IF state = 0 OR state = 9 THEN
	IF Busy THEN
		LastExecutionResult.Done := Done;
		LastExecutionResult.CommandAborted := CommandAborted;
		LastExecutionResult.Error := Error;
		LastExecutionResult.ErrorID := ErrorID;
	END_IF
	Busy := FALSE;
	Active := FALSE;
ELSIF F_AxisInProtectedMode(Axis.NcToPlc.StateDWord) THEN (* 2009-11-18 KSt *)
	(* if axis is coupled on the fly - force state machine back to state zero and signal an error *)
	state := 0;
	Error := TRUE;
	ErrorID := MC_ERROR_AXIS_IN_PROTECTED_MODE;
END_IF
END_FUNCTION_BLOCK
ACTION ActCheckJogEnd:
JogEnd := 	(NOT JogForward AND NOT JogBackwards) OR
			(NOT JogForward AND Direction=MC_Positive_Direction) OR
			(NOT JogBackwards AND Direction=MC_Negative_Direction);
END_ACTION
ACTION ActJogMove:
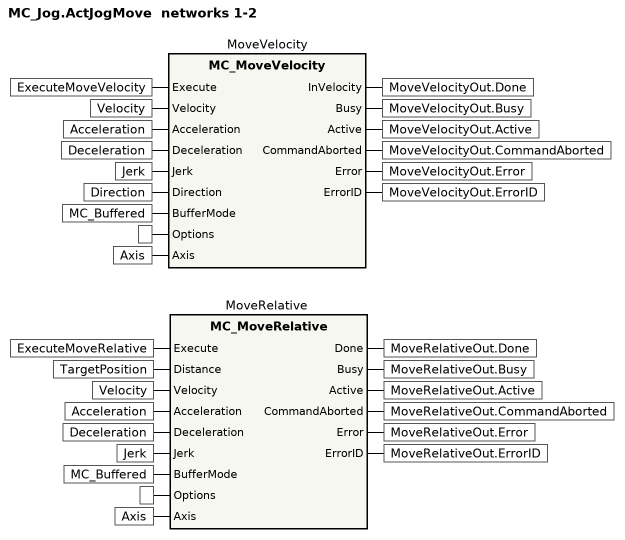
[picture p9: MC_Jog.ActJogMove (FBD) networks 1-2]
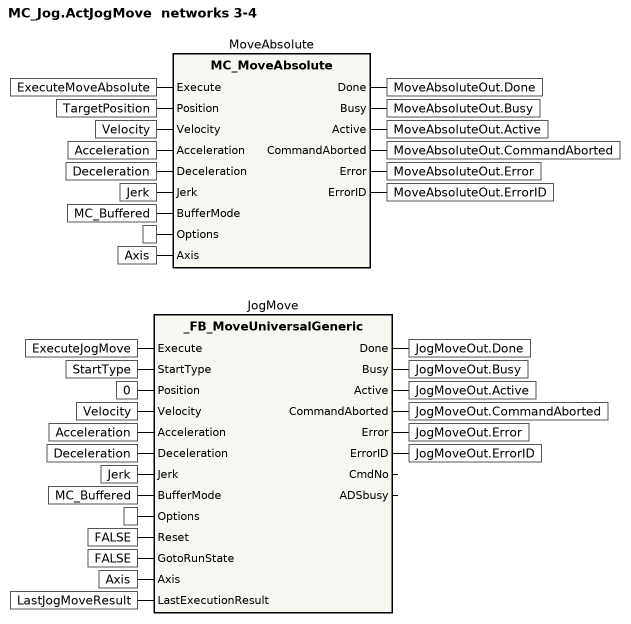
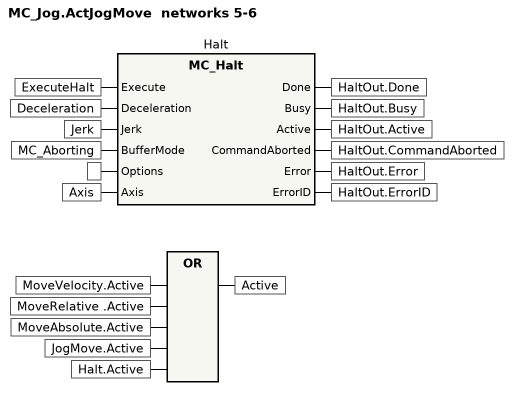
_FBD_ (* Function Block Diagram *)
NETWORK 1
	MoveVelocity:MC_MoveVelocity(Execute: ExecuteMoveVelocity, Velocity: Velocity, Acceleration: Acceleration, Deceleration: Deceleration, Jerk: Jerk, Direction: Direction, BufferMode: MC_Buffered, Options: , Axis: Axis, Busy => MoveVelocityOut.Busy, Active => MoveVelocityOut.Active, CommandAborted => MoveVelocityOut.CommandAborted, Error => MoveVelocityOut.Error, ErrorID => MoveVelocityOut.ErrorID) => MoveVelocityOut.Done
NETWORK 2
	MoveRelative :MC_MoveRelative(Execute: ExecuteMoveRelative, Distance: TargetPosition, Velocity: Velocity, Acceleration: Acceleration, Deceleration: Deceleration, Jerk: Jerk, BufferMode: MC_Buffered, Options: , Axis: Axis, Busy => MoveRelativeOut.Busy, Active => MoveRelativeOut.Active, CommandAborted => MoveRelativeOut.CommandAborted, Error => MoveRelativeOut.Error, ErrorID => MoveRelativeOut.ErrorID) => MoveRelativeOut.Done
NETWORK 3
	MoveAbsolute:MC_MoveAbsolute(Execute: ExecuteMoveAbsolute, Position: TargetPosition, Velocity: Velocity, Acceleration: Acceleration, Deceleration: Deceleration, Jerk: Jerk, BufferMode: MC_Buffered, Options: , Axis: Axis, Busy => MoveAbsoluteOut.Busy, Active => MoveAbsoluteOut.Active, CommandAborted => MoveAbsoluteOut.CommandAborted, Error => MoveAbsoluteOut.Error, ErrorID => MoveAbsoluteOut.ErrorID) => MoveAbsoluteOut.Done
NETWORK 4
	JogMove:_FB_MoveUniversalGeneric(Execute: ExecuteJogMove, StartType: StartType, Position: 0, Velocity: Velocity, Acceleration: Acceleration, Deceleration: Deceleration, Jerk: Jerk, BufferMode: MC_Buffered, Options: , Reset: FALSE, GotoRunState: FALSE, Axis: Axis, LastExecutionResult: LastJogMoveResult, Busy => JogMoveOut.Busy, Active => JogMoveOut.Active, CommandAborted => JogMoveOut.CommandAborted, Error => JogMoveOut.Error, ErrorID => JogMoveOut.ErrorID) => JogMoveOut.Done
NETWORK 5
	Halt:MC_Halt(Execute: ExecuteHalt, Deceleration: Deceleration, Jerk: Jerk, BufferMode: MC_Aborting, Options: , Axis: Axis, Busy => HaltOut.Busy, Active => HaltOut.Active, CommandAborted => HaltOut.CommandAborted, Error => HaltOut.Error, ErrorID => HaltOut.ErrorID) => HaltOut.Done
NETWORK 6
	OR(MoveVelocity.Active, MoveRelative .Active, MoveAbsolute.Active, JogMove.Active, Halt.Active) => Active
_END_FBD_
(* the same logic as Structured Text *)
(* Network 1: see the listing above *)
(* Network 2: see the listing above *)
(* Network 3: see the listing above *)
(* Network 4: see the listing above *)
(* Network 5: see the listing above *)
(* Network 6 *)
Active := MoveVelocity.Active OR (MoveRelative .Active) OR MoveAbsolute.Active OR JogMove.Active OR Halt.Active;
END_ACTION

(* POU MC_MoveVelocity, FBD *)
FUNCTION_BLOCK MC_MoveVelocity
(*	This Function Block commands a never ending controlled motion at a specified velocity. *)
VAR_IN_OUT
	Axis				:	AXIS_REF;	(* B *)
END_VAR
VAR_INPUT
	Execute			:	BOOL;	(* B *)
(*	ContinuousUpdate :	BOOL; *)	(* E *)	(* not available *)
	Velocity			:	LREAL;	(* E *)
	Acceleration		:	LREAL;	(* E *)
	Deceleration		:	LREAL;	(* E *)
	Jerk				:	LREAL;	(* E *)
	Direction			:	MC_Direction := MC_Positive_Direction;	(* E *)
	BufferMode		:	MC_BufferMode;	(* E *)
	Options			: 	ST_MoveOptions; (* V *)
END_VAR
VAR_OUTPUT
	InVelocity		:	BOOL;	(* B *)	(* Commanded velocity reached *)
	Busy			: 	BOOL;	(* E *)
	Active			: 	BOOL;	(* E *)
	CommandAborted	:	BOOL;	(* E *)
	Error			:	BOOL;	(* B *)
	ErrorID			:	UDINT;	(* E *)
END_VAR
VAR
	LastExecutionResult: 	_ST_FunctionBlockResults;
	ADSbusy		: 	BOOL;
	MoveGeneric		: 	_FB_MoveUniversalGeneric;
	CmdNo: UINT;
END_VAR
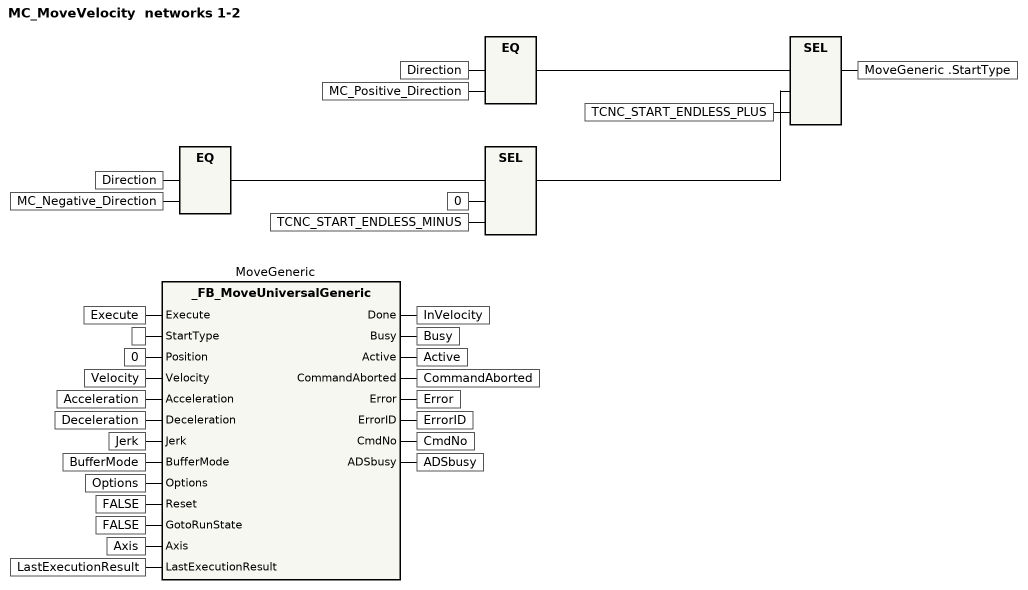
_FBD_ (* Function Block Diagram *)
NETWORK 1
	SEL(EQ(Direction, MC_Positive_Direction), SEL(EQ(Direction, MC_Negative_Direction), 0, TCNC_START_ENDLESS_MINUS), TCNC_START_ENDLESS_PLUS) => MoveGeneric .StartType
NETWORK 2
	MoveGeneric   :_FB_MoveUniversalGeneric(Execute: Execute, StartType: , Position: 0, Velocity: Velocity, Acceleration: Acceleration, Deceleration: Deceleration, Jerk: Jerk, BufferMode: BufferMode, Options: Options, Reset: FALSE, GotoRunState: FALSE, Axis: Axis, LastExecutionResult: LastExecutionResult, Busy => Busy, Active => Active, CommandAborted => CommandAborted, Error => Error, ErrorID => ErrorID, CmdNo => CmdNo, ADSbusy => ADSbusy) => InVelocity
_END_FBD_
(* the same logic as Structured Text *)
(* Network 1 *)
MoveGeneric .StartType := SEL(Direction = MC_Positive_Direction, SEL(Direction = MC_Negative_Direction, 0, TCNC_START_ENDLESS_MINUS), TCNC_START_ENDLESS_PLUS);
(* Network 2: see the listing above *)
END_FUNCTION_BLOCK

(* POU MC_MoveRelative, FBD *)
FUNCTION_BLOCK MC_MoveRelative
(*	This Function Block commands a controlled motion of a specified distance
	relative to the actual position at the time of the execution.
*)
VAR_IN_OUT
	Axis				:	AXIS_REF;	(* B *)
END_VAR
VAR_INPUT
	Execute			:	BOOL;	(* B *)
(*	ContinuousUpdate :	BOOL; *)	(* E *)	(* not available *)
	Distance			:	LREAL;	(* B *)
	Velocity			:	LREAL;	(* E *)
	Acceleration		:	LREAL;	(* E *)
	Deceleration		:	LREAL;	(* E *)
	Jerk				:	LREAL;	(* E *)
	BufferMode		:	MC_BufferMode;	(* E *)
	Options			: 	ST_MoveOptions;	(* V *)
END_VAR
VAR_OUTPUT
	Done			:	BOOL;	(* B *)
	Busy			: 	BOOL;	(* E *)
	Active			: 	BOOL;	(* E *)
	CommandAborted	:	BOOL;	(* E *)
	Error			:	BOOL;	(* B *)
	ErrorID			:	UDINT;	(* E *)
END_VAR
VAR
	LastExecutionResult: 	_ST_FunctionBlockResults;
	ADSbusy		: 	BOOL;
	MoveGeneric		: 	_FB_MoveUniversalGeneric;
	CmdNo: UINT;
END_VAR
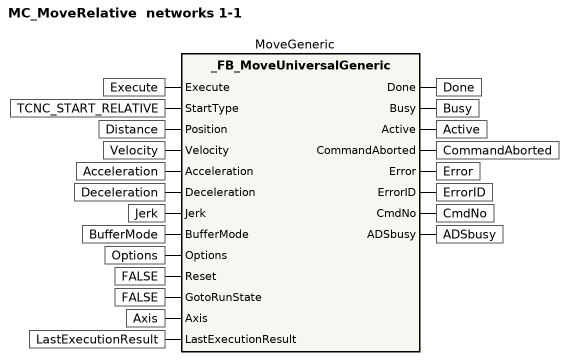
_FBD_ (* Function Block Diagram *)
NETWORK 1
	MoveGeneric   :_FB_MoveUniversalGeneric(Execute: Execute, StartType: TCNC_START_RELATIVE, Position: Distance, Velocity: Velocity, Acceleration: Acceleration, Deceleration: Deceleration, Jerk: Jerk, BufferMode: BufferMode, Options: Options, Reset: FALSE, GotoRunState: FALSE, Axis: Axis, LastExecutionResult: LastExecutionResult, Busy => Busy, Active => Active, CommandAborted => CommandAborted, Error => Error, ErrorID => ErrorID, CmdNo => CmdNo, ADSbusy => ADSbusy) => Done
_END_FBD_
(* the same logic as Structured Text *)
(* Network 1 *)
MoveGeneric   (Execute := Execute, StartType := TCNC_START_RELATIVE, Position := Distance, Velocity := Velocity, Acceleration := Acceleration, Deceleration := Deceleration, Jerk := Jerk, BufferMode := BufferMode, Options := Options, Reset := FALSE, GotoRunState := FALSE, Axis := Axis, LastExecutionResult := LastExecutionResult);
Busy := MoveGeneric   .Busy;
Active := MoveGeneric   .Active;
CommandAborted := MoveGeneric   .CommandAborted;
Error := MoveGeneric   .Error;
ErrorID := MoveGeneric   .ErrorID;
CmdNo := MoveGeneric   .CmdNo;
ADSbusy := MoveGeneric   .ADSbusy;
Done := MoveGeneric   .Done;
END_FUNCTION_BLOCK

(* POU MC_MoveAdditive, FBD *)
FUNCTION_BLOCK MC_MoveAdditive
(*	This Function Block commands a controlled motion of a specified relative
	distance additional to the most recent commanded position in the discrete 
	motion state. The most recent commanded position may be the result of a 
	previous MC_MoveAdditive motion which was aborted. If the FB is activated 
	in the Continuous Mode the specified relative distance is added to the actual 
	position at the time of the execution.

 	MC_MoveAdditive ist ähnlich MC_MoveRelative. Wenn während der Bewegung
	getriggert, dann wird allerdings die ursprüngliche Zielposition um Distance 
	verlängert. Eine Endlosachse wird in eine diskrete Bewegung ausgehend 
	von der aktuellen Position plus Distanz gewandelt.
*)
VAR_IN_OUT
	Axis				:	AXIS_REF; (* B *)
END_VAR
VAR_INPUT
	Execute			:	BOOL;	(* B *)
(*	ContinuousUpdate :	BOOL; *)	(* E *)	(* not available *)
	Distance			:	LREAL;	(* B *)
	Velocity			:	LREAL;	(* E *)
	Acceleration		:	LREAL;	(* E *)
	Deceleration		:	LREAL;	(* E *)
	Jerk				:	LREAL;	(* E *)
	BufferMode		:	MC_BufferMode;	(* E *)
	Options			: 	ST_MoveOptions;	(* V *)
END_VAR
VAR_OUTPUT
	Done			:	BOOL;	(* B *)
	Busy			: 	BOOL;	(* E *)
	Active			: 	BOOL;	(* E *)
	CommandAborted	:	BOOL;	(* E *)
	Error			:	BOOL;	(* B *)
	ErrorID			:	UDINT;	(* E *)
END_VAR
VAR
	LastExecutionResult: 	_ST_FunctionBlockResults;
	ADSbusy		: 	BOOL;
	MoveGeneric		: 	_FB_MoveUniversalGeneric;
	CmdNo: UINT;
END_VAR
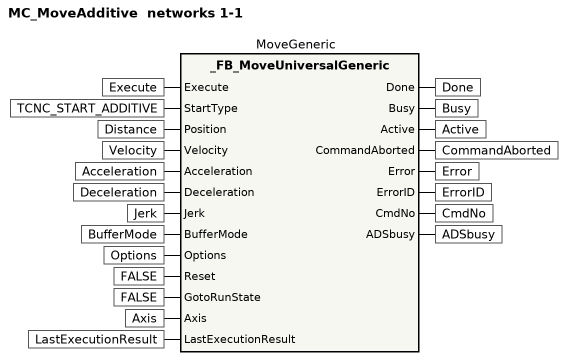
_FBD_ (* Function Block Diagram *)
NETWORK 1
	MoveGeneric  :_FB_MoveUniversalGeneric(Execute: Execute, StartType: TCNC_START_ADDITIVE, Position: Distance, Velocity: Velocity, Acceleration: Acceleration, Deceleration: Deceleration, Jerk: Jerk, BufferMode: BufferMode, Options: Options, Reset: FALSE, GotoRunState: FALSE, Axis: Axis, LastExecutionResult: LastExecutionResult, Busy => Busy, Active => Active, CommandAborted => CommandAborted, Error => Error, ErrorID => ErrorID, CmdNo => CmdNo, ADSbusy => ADSbusy) => Done
_END_FBD_
(* the same logic as Structured Text *)
(* Network 1 *)
MoveGeneric  (Execute := Execute, StartType := TCNC_START_ADDITIVE, Position := Distance, Velocity := Velocity, Acceleration := Acceleration, Deceleration := Deceleration, Jerk := Jerk, BufferMode := BufferMode, Options := Options, Reset := FALSE, GotoRunState := FALSE, Axis := Axis, LastExecutionResult := LastExecutionResult);
Busy := MoveGeneric  .Busy;
Active := MoveGeneric  .Active;
CommandAborted := MoveGeneric  .CommandAborted;
Error := MoveGeneric  .Error;
ErrorID := MoveGeneric  .ErrorID;
CmdNo := MoveGeneric  .CmdNo;
ADSbusy := MoveGeneric  .ADSbusy;
Done := MoveGeneric  .Done;
END_FUNCTION_BLOCK

(* POU MC_MoveContinuousAbsolute, FBD *)
FUNCTION_BLOCK MC_MoveContinuousAbsolute
(*	This function block commands a controlled motion to a specified absolute position
	ending with the specified velocity.

	Notes:
	- If the target is reached and no new motion command is put into the buffer, the 
	  axis continues to run with the specified ‘EndVelocity’.
	- This Function Block places the axis into the 'Continuous Motion' state, even 
	  during the initial motion by a relative distance, and remains in the 'Continuous 
	  Motion' state once the EndVelocity has been reached.
	- This FB can be replaced by the combination of MC_MoveAbsolute and 
	  MC_MoveVelocity

	MoveContinous ist ähnlich MoveVelocity. Es wird aber zunächst mit einem PTP-Profil
	eine Zwischenposition angefahren (mit Velocity). Ab dieser Position geht die Bewegung
	in eine Endlosfahrt mit EndVelocity über.
*)
VAR_IN_OUT
	Axis				:	AXIS_REF; (* B *)
END_VAR
VAR_INPUT
	Execute			:	BOOL;	(* B *)
(*	ContinuousUpdate :	BOOL; *)	(* E *)	(* not available *)
	Position			:	LREAL;	(* B *)
	Velocity			:	LREAL;	(* B *)
	EndVelocity		:	LREAL;	(* B *)
	Acceleration		:	LREAL;	(* E *)
	Deceleration		:	LREAL;	(* E *)
	Jerk				:	LREAL;	(* E *)
(*	Direction 		:	MC_Direction;	*)	(* E *)	(* not available *)
	BufferMode		:	MC_BufferMode;	(* E *)
	Options			: 	ST_MoveOptions;
END_VAR
VAR_OUTPUT
	InEndVelocity		:	BOOL;	(* B *)
	Busy			: 	BOOL;	(* E *)
	Active			: 	BOOL;	(* E *)
	CommandAborted :	BOOL;	(* E *)
	Error			:	BOOL;	(* B *)
	ErrorID			:	UDINT;	(* E *)
END_VAR
VAR
	LastExecutionResult: 	_ST_FunctionBlockResults;
	ADSbusy		: 	BOOL;
	MoveGeneric		: 	_FB_MoveUniversalGeneric;
	CmdNo: UINT;
END_VAR
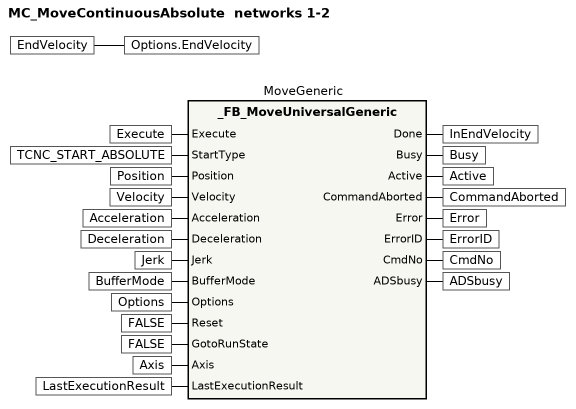
_FBD_ (* Function Block Diagram *)
NETWORK 1
	EndVelocity => Options.EndVelocity
NETWORK 2
	MoveGeneric  :_FB_MoveUniversalGeneric(Execute: Execute, StartType: TCNC_START_ABSOLUTE, Position: Position, Velocity: Velocity, Acceleration: Acceleration, Deceleration: Deceleration, Jerk: Jerk, BufferMode: BufferMode, Options: Options, Reset: FALSE, GotoRunState: FALSE, Axis: Axis, LastExecutionResult: LastExecutionResult, Busy => Busy, Active => Active, CommandAborted => CommandAborted, Error => Error, ErrorID => ErrorID, CmdNo => CmdNo, ADSbusy => ADSbusy) => InEndVelocity
_END_FBD_
(* the same logic as Structured Text *)
(* Network 1 *)
Options.EndVelocity := EndVelocity;
(* Network 2 *)
MoveGeneric  (Execute := Execute, StartType := TCNC_START_ABSOLUTE, Position := Position, Velocity := Velocity, Acceleration := Acceleration, Deceleration := Deceleration, Jerk := Jerk, BufferMode := BufferMode, Options := Options, Reset := FALSE, GotoRunState := FALSE, Axis := Axis, LastExecutionResult := LastExecutionResult);
Busy := MoveGeneric  .Busy;
Active := MoveGeneric  .Active;
CommandAborted := MoveGeneric  .CommandAborted;
Error := MoveGeneric  .Error;
ErrorID := MoveGeneric  .ErrorID;
CmdNo := MoveGeneric  .CmdNo;
ADSbusy := MoveGeneric  .ADSbusy;
InEndVelocity := MoveGeneric  .Done;
END_FUNCTION_BLOCK

(* POU MC_MoveContinuousRelative, FBD *)
FUNCTION_BLOCK MC_MoveContinuousRelative
(*	This function block commands a controlled motion of a specified relative distance
	ending with the specified velocity.

	Notes:
	- If the target is reached and no new motion command is put into the buffer, the 
	  axis continues to run with the specified ‘EndVelocity’.
	- This Function Block places the axis into the 'Continuous Motion' state, even 
	  during the initial motion by a relative distance, and remains in the 'Continuous 
	  Motion' state once the EndVelocity has been reached.
 	- This FB can be replaced by the combination of MC_MoveRelative and 
	  MC_MoveVelocity 

	MoveContinous ist ähnlich MoveVelocity. Es wird aber zunächst mit einem PTP-Profil
	eine Zwischenposition angefahren (mit Velocity). Ab dieser Position geht die Bewegung
	in eine Endlosfahrt mit EndVelocity über.
*)
VAR_IN_OUT
	Axis				:	AXIS_REF; (* B *)
END_VAR
VAR_INPUT
	Execute			:	BOOL;	(* B *)
(*	ContinuousUpdate :	BOOL; *)	(* E *)	(* not available *)
	Distance			:	LREAL;	(* B *)
	Velocity			:	LREAL;	(* B *)
	EndVelocity		:	LREAL;	(* B *)
	Acceleration		:	LREAL;	(* E *)
	Deceleration		:	LREAL;	(* E *)
	Jerk				:	LREAL;	(* E *)
	BufferMode		:	MC_BufferMode;	(* E *)
	Options			: 	ST_MoveOptions;
END_VAR
VAR_OUTPUT
	InEndVelocity		:	BOOL;	(* B *)
	Busy			: 	BOOL;	(* E *)
	Active			: 	BOOL;	(* E *)
	CommandAborted :	BOOL;	(* E *)
	Error			:	BOOL;	(* B *)
	ErrorID			:	UDINT;	(* E *)
END_VAR
VAR
	LastExecutionResult: 	_ST_FunctionBlockResults;
	ADSbusy		: 	BOOL;
	MoveGeneric		: 	_FB_MoveUniversalGeneric;
	CmdNo: UINT;
END_VAR
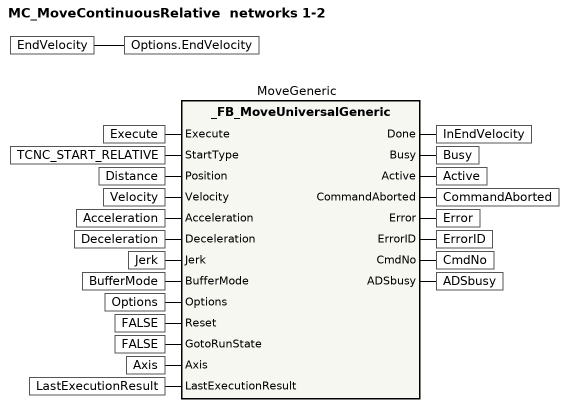
_FBD_ (* Function Block Diagram *)
NETWORK 1
	EndVelocity => Options.EndVelocity
NETWORK 2
	MoveGeneric  :_FB_MoveUniversalGeneric(Execute: Execute, StartType: TCNC_START_RELATIVE, Position: Distance, Velocity: Velocity, Acceleration: Acceleration, Deceleration: Deceleration, Jerk: Jerk, BufferMode: BufferMode, Options: Options, Reset: FALSE, GotoRunState: FALSE, Axis: Axis, LastExecutionResult: LastExecutionResult, Busy => Busy, Active => Active, CommandAborted => CommandAborted, Error => Error, ErrorID => ErrorID, CmdNo => CmdNo, ADSbusy => ADSbusy) => InEndVelocity
_END_FBD_
(* the same logic as Structured Text *)
(* Network 1 *)
Options.EndVelocity := EndVelocity;
(* Network 2 *)
MoveGeneric  (Execute := Execute, StartType := TCNC_START_RELATIVE, Position := Distance, Velocity := Velocity, Acceleration := Acceleration, Deceleration := Deceleration, Jerk := Jerk, BufferMode := BufferMode, Options := Options, Reset := FALSE, GotoRunState := FALSE, Axis := Axis, LastExecutionResult := LastExecutionResult);
Busy := MoveGeneric  .Busy;
Active := MoveGeneric  .Active;
CommandAborted := MoveGeneric  .CommandAborted;
Error := MoveGeneric  .Error;
ErrorID := MoveGeneric  .ErrorID;
CmdNo := MoveGeneric  .CmdNo;
ADSbusy := MoveGeneric  .ADSbusy;
InEndVelocity := MoveGeneric  .Done;
END_FUNCTION_BLOCK

(* POU MC_MoveModulo, ST *)
FUNCTION_BLOCK MC_MoveModulo
(* This Function Block commands a controlled motion to a specified absolute modulo position. *)
VAR_IN_OUT
	Axis				:	AXIS_REF;
END_VAR
VAR_INPUT
	Execute			:	BOOL;
	Position			:	LREAL;
	Velocity			:	LREAL;
	Acceleration		:	LREAL;
	Deceleration		:	LREAL;
	Jerk				:	LREAL;
	Direction			:	MC_Direction;	(* E *)	(* modulo shortest way, modulo positive, modulo negative *)
	BufferMode		:	MC_BufferMode;(* E *)
	Options			: 	ST_MoveOptions;
END_VAR
VAR_OUTPUT
	Done				:	BOOL;	(* B *)
	Busy				: 	BOOL;	(* E *)
	Active				: 	BOOL;	(* E *)
	CommandAborted		:	BOOL;	(* E *)
	Error				:	BOOL;	(* B *)
	ErrorID				:	UDINT;	(* E *)
END_VAR
VAR
	LastExecutionResult: _ST_FunctionBlockResults;
	ADSbusy: BOOL;
	MoveGeneric: _FB_MoveUniversalGeneric;
(*	StartType: UDINT;*)
	StartType: _E_TcNC_StartPosType;	(* 20110511 KSt type changed for TC3 *)
	CmdNo: UINT;
END_VAR
{ library private }
VAR
	TriggerExecute: R_TRIG;
END_VAR
(*  new move modulo code - KST 2012-03-23 *)
TriggerExecute(CLK:=Execute);
IF TriggerExecute.Q AND NOT MoveGeneric.Busy THEN
	(* initialize the start type when block is triggered *)
	CASE Direction OF
		MC_Positive_Direction:
			StartType := TCNC_START_MODULO_PLUS;
		MC_Shortest_Way:
			StartType := TCNC_START_MODULO_SHORT;
		MC_Negative_Direction:
			StartType := TCNC_START_MODULO_MINUS;
		MC_Current_Direction:
			StartType := TCNC_START_MODULO_CURRENT;
		ELSE
			StartType := 0; (* set to undefined *)
			Error := TRUE;
			ErrorID := MC_ERROR_WRONG_MODE;
			Done := FALSE;
			Busy := FALSE;
			Active := FALSE;
			CommandAborted := FALSE;
			(* generic move block will not be called *)
	END_CASE
END_IF

IF StartType<>0 THEN
	(* just call the generic move block *)
	MC_MoveModuloCall();
END_IF


(* old code before 2012-03-23 - KST *)
(*
CASE Direction OF
	MC_Positive_Direction:
		StartType := TCNC_START_MODULO_PLUS;
		MC_MoveModuloCall;

	MC_Shortest_Way:
		StartType := TCNC_START_MODULO_SHORT;
		MC_MoveModuloCall;

	MC_Negative_Direction:
		StartType := TCNC_START_MODULO_MINUS;
		MC_MoveModuloCall;

	MC_Current_Direction:
		StartType := TCNC_START_MODULO_CURRENT;
		MC_MoveModuloCall;
	ELSE
		IF Execute THEN
			Error := TRUE;
			ErrorID := MC_ERROR_WRONG_MODE;
		ELSE
			Error := FALSE;
			ErrorID := 0;
		END_IF
		Execute := FALSE;
		MC_MoveModuloCall;
		Done := FALSE;
		Busy := FALSE;
		Active := FALSE;
		CommandAborted := FALSE;
END_CASE
*)
END_FUNCTION_BLOCK
ACTION MC_MoveModuloCall:
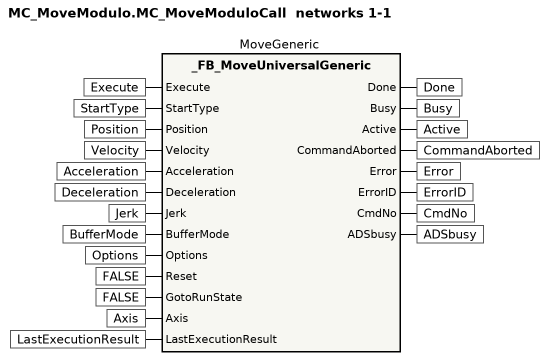
_FBD_ (* Function Block Diagram *)
NETWORK 1
	MoveGeneric :_FB_MoveUniversalGeneric(Execute: Execute, StartType: StartType, Position: Position, Velocity: Velocity, Acceleration: Acceleration, Deceleration: Deceleration, Jerk: Jerk, BufferMode: BufferMode, Options: Options, Reset: FALSE, GotoRunState: FALSE, Axis: Axis, LastExecutionResult: LastExecutionResult, Busy => Busy, Active => Active, CommandAborted => CommandAborted, Error => Error, ErrorID => ErrorID, CmdNo => CmdNo, ADSbusy => ADSbusy) => Done
_END_FBD_
(* the same logic as Structured Text *)
(* Network 1 *)
MoveGeneric (Execute := Execute, StartType := StartType, Position := Position, Velocity := Velocity, Acceleration := Acceleration, Deceleration := Deceleration, Jerk := Jerk, BufferMode := BufferMode, Options := Options, Reset := FALSE, GotoRunState := FALSE, Axis := Axis, LastExecutionResult := LastExecutionResult);
Busy := MoveGeneric .Busy;
Active := MoveGeneric .Active;
CommandAborted := MoveGeneric .CommandAborted;
Error := MoveGeneric .Error;
ErrorID := MoveGeneric .ErrorID;
CmdNo := MoveGeneric .CmdNo;
ADSbusy := MoveGeneric .ADSbusy;
Done := MoveGeneric .Done;
END_ACTION

(* POU MC_MoveSuperImposed, ST *)
(*	MC_MovedSuperimposed	(extended version 2)

	This Function Block commands a controlled motion of a specified relative distance additional to an existing motion.
	The existing Motion is not interrupted, but is superimposed by the additional motion.

	- Version 2 adds multiple modes and feedback information to the 
	  standard MC_MoveSuperimposed block.
 	- The version 2 block is compatible to the MC_MovedSuperimposed block when Mode
	  SUPERPOSITIONMODE_VELOREDUCTION_ADDITIVEMOTION (integer value 1) is used.

	The values of ‘Acceleration’, ‘Deceleration’, and ‘Jerk’ are additional values to the on-going motion, and not
	absolute ones. With this, the underlying FB always finishes its job in the same period of time regardless of
	whether a MC_MoveSuperimposed FB takes place concurrently.
 *)
FUNCTION_BLOCK MC_MoveSuperImposed
VAR_IN_OUT
	Axis				:	AXIS_REF;	(* B *)
END_VAR
VAR_INPUT
	Execute			:	BOOL;	(* B *)
	Mode 			:	E_SuperpositionMode;	(* V *)
(*	ContinuousUpdate :	BOOL; *)	(* E *)	(* not available *)
	Distance			:	LREAL;	(* B *)	(* distance to catch up or fall back with the superposition process *)
	VelocityDiff		:	LREAL;	(* E *)	(* maximum velocity difference - will be added or subtrated to the process velocity *)
	Acceleration		:	LREAL;	(* E *)
	Deceleration		:	LREAL;	(* E *)
	Jerk				:	LREAL;	(* E *)	(* currently not used *)
	VelocityProcess	:	LREAL;	(* V *)	(* constant velocity of the axis without superposition *)
	Length			:	LREAL;	(* V *)	(* moved distance while the superposition takes place (name has been MaxDistance before) *)
	Options			:	ST_SuperpositionOptions;	(* V *)
END_VAR
VAR_OUTPUT
	Done			:	BOOL;	(* B *)
	Busy			:	BOOL;	(* E *)
	Active			:	BOOL;	(* E *)
	CommandAborted	:	BOOL;	(* E *)
	Error			:	BOOL;	(* B *)
	ErrorID			:	UDINT;	(* E *)
(*	CoveredDistance	:	LREAL;*)	(* E *)	(* not available *)
	Warning			: 	BOOL;	(* V *)
	WarningId		: 	UDINT;	(* V *)
	ActualVelocityDiff	: 	LREAL;	(* V *)	(* calculated maximum velocity boost during superposition <= VelocityDiff *)
	ActualDistance	: 	LREAL;	(* V *)	(* calculated superimposed distance <= Distance*)
	ActualLength		: 	LREAL;	(* V *)	(* calculated length of the superposition <= MaxDistance *)
	ActualAcceleration : 	LREAL;	(* V *)	(* calculated acceleration during superposition *)
	ActualDeceleration : 	LREAL;	(* V *)	(* calculated deceleration during superposition *)
END_VAR
VAR
	LastExecutionResult: 	_ST_FunctionBlockResults;
	ADSbusy		: 	BOOL;
	CompensationStarted: 	BOOL;
	AxisHasJobAtStartOfCompensation	: 	BOOL; 	(* HasJob flag when starting the compensation *)
	AxisIsMovingAtStartOfCompensation	:	BOOL; 	(* Moving flag when starting the compensation *)
	iState			: 	_E_TcMC_STATES := STATE_INITIALIZATION;
	fbAdsReadWrite	: 	ADSRDWRTEX;
	sNcCompensation	:	_ST_TcNC_Compensation2;
END_VAR
{library private}
VAR
	fbTrigger			:	R_TRIG;
	fbTimeOut		: 	TON;
END_VAR
(* ====================================================================== *)
(* *)
(* ====================================================================== *)
fbTrigger(CLK:= Execute);

CASE iState OF
STATE_INITIALIZATION:	(* *)
	Busy := FALSE;
	Active := FALSE;

	IF NOT Execute THEN
		Done := FALSE;
		CommandAborted := FALSE;
		Error := FALSE;			(* reset at falling edge of Execute *)
		ErrorID := 0;
	END_IF;

    	IF fbTrigger.Q THEN
		(* initialize output values *)
		Done := FALSE;
		Busy := TRUE;
		CommandAborted := FALSE;
		Error := FALSE;
		ErrorID := 0;
		Warning := FALSE;
		WarningId := 0;
		LastExecutionResult.Done := FALSE;
		LastExecutionResult.CommandAborted := FALSE;
		LastExecutionResult.Error := FALSE;
		LastExecutionResult.ErrorID := 0;
		ActualVelocityDiff := 0;
		ActualDistance := 0;
		ActualLength := 0;
		CompensationStarted := FALSE;
		fbTimeOut(IN:= FALSE);
		fbAdsReadWrite(WRTRD:=FALSE);

		(* 2009-10-06 KSt - initial HasJob and InMotion state check *)
		AxisHasJobAtStartOfCompensation := F_AxisHasJob(Axis.NcToPlc.StateDWord);
		AxisIsMovingAtStartOfCompensation := F_AxisIsMoving(Axis.NcToPlc.StateDWord);
		(* error when ... *)
		(* 24.09.2009 HKP - Fehlerabfrage nur im Default-Fall mit  '(0) SUPERPOSITIONOPTION_ABORTATSTANDSTILL' sinnvoll *)
		(* IF  NOT F_AxisHasJob(Axis.NcToPlc.StateDWord) THEN  *) (* 12.6.2007 KSt - geändert von "NOT AxisIsMoving" nach "NOT AxisHasJob" *)
		IF  Options.AbortOption = SUPERPOSITIONOPTION_ABORTATSTANDSTILL AND NOT  F_AxisHasJob(Axis.NcToPlc.StateDWord) THEN
			ErrorID := MC_ERROR_AXIS_IS_NOT_MOVING;
			Error := TRUE;
		ELSE
			(* fill structure *)
			sNcCompensation.nCompType		:= Mode;
			sNcCompensation.fAccPlus			:= Acceleration;
			sNcCompensation.fAccMinus		:= Deceleration;
			sNcCompensation.fVeloDiff			:= VelocityDiff;
			sNcCompensation.fVeloProcess		:= VelocityProcess;
			sNcCompensation.fDistance		:= Distance;
			sNcCompensation.fLength		 	:= Length;
			(* WarningID holds optional parameters when sending the command to the NC *)
			sNcCompensation.nWarningId		:= Options.AbortOption; (* 2009-06-30 KSt *)

			(* fbAdsReadWrite.PORT := SEL(Axis.ADS.Port = 0, Axis.ADS.port, AMSPORT_R0_NCSAF);*)				(* KSt, 20140930 *)
			fbAdsReadWrite.PORT := SEL(Axis.ADS.Port = 0, Axis.ADS.port, TcMcGlobal.NCPORT_TCMC_SUPERPOSITION);	(* KSt, 20140930 *)
			fbAdsReadWrite(NETID:= TcMcGlobal.NCNETID_TCMC,
							(* PORT:= TcMcGlobal.NCPORT_TCMC,*) 		(* KSt, 20090123 *)
							IDXGRP:= TcMcGlobal.Axis.Functions.IDXGRP+Axis.NcToPlc.AxisId,
							IDXOFFS:= TcMcGlobal.Axis.Functions.IDXOFFS.STARTSCOM,
							WRITELEN:= SIZEOF(sNcCompensation),
							READLEN:= SIZEOF(sNcCompensation),
							SRCADDR:= ADR(sNcCompensation),
							DESTADDR:= ADR(sNcCompensation),
							WRTRD:= TRUE,
							TMOUT:= TcMcGlobal.tADSTimeOut );

			iState := STATE_ORDER;
		END_IF;
	END_IF;

STATE_ORDER:  (* wait until command is accepted *)
	fbAdsReadWrite(WRTRD:= TRUE);
	IF NOT fbAdsReadWrite.Busy THEN
		IF fbAdsReadWrite.Err THEN
			Error := TRUE;
			ErrorID := fbAdsReadWrite.ErrId;
			iState := STATE_INITIALIZATION;
		ELSE
			IF fbAdsReadWrite.COUNT_R > 0 THEN
				ActualVelocityDiff := sNcCompensation.fVeloDiff;
				ActualDistance := sNcCompensation.fDistance;
				ActualLength := sNcCompensation.fLength;
				ActualAcceleration := sNcCompensation.fAccPlus;		(* 2010-02-25 KSt *)
				ActualDeceleration := sNcCompensation.fAccMinus;	(* 2010-02-25 KSt *)
				WarningId := sNcCompensation.nWarningId;	(* 2009-01-29 KSt *)
				Warning := WarningId <> 0;					(* 2009-01-29 KSt *)
			END_IF
			Active := TRUE;
			CompensationStarted := F_AxisIsCompensating(Axis.NcToPlc.StateDWord) ;
			iState := STATE_RUNNING;
		END_IF;
	END_IF;

STATE_RUNNING:  (* wait until axis stands still *)
	WarningId := sNcCompensation.nWarningId;
	Warning := WarningId <> 0;
(*	Busy := F_AxisIsCompensating(Axis.NcToPlc.StateDWord);
	IF Busy THEN	KSt, 29.4.2008 *)

	IF F_AxisIsCompensating(Axis.NcToPlc.StateDWord) THEN 	(* KSt, 29.4.2008 *)
		CompensationStarted := TRUE;
	ELSIF CompensationStarted  (* AND compensation finished now *) THEN
		IF AxisHasJobAtStartOfCompensation AND NOT F_AxisHasJob(Axis.NcToPlc.StateDWord) THEN (* 2009-10-06 KSt *)
			(* command aborted, move has been stopped before superposition finished because the HasJob flag turned off (KSt, 2009-08-13) *)
			CommandAborted := TRUE;
			iState := STATE_INITIALIZATION;
		ELSIF NOT AxisHasJobAtStartOfCompensation AND AxisIsMovingAtStartOfCompensation THEN (* 2009-10-06 KSt *)
			(* in case of axes coupled to actual position (encoder axes or disabled axes) *)
			IF NOT F_AxisIsMoving(Axis.NcToPlc.StateDWord) THEN (* 2009-10-06 KSt *)
				CommandAborted := TRUE;
				iState := STATE_INITIALIZATION;
			ELSE
				(* check moving state next cycle - delay is necessary since moving flag turnes off later than the compensation flag *)
				iState := STATE_WAITING;
			END_IF
		ELSE
			(* the initial HasJob or Moving state was the same as at end of compensation - assume that superposition completed *)
			Done := TRUE;
			iState := STATE_INITIALIZATION;
		END_IF
	ELSE (* compensation did not start so far *)
		(* check for superposition not beeing started (KSt, 12.01.2004) *)
		fbTimeOut(IN:= TRUE, PT:= T#50ms);
		IF fbTimeOut.Q THEN
			(*	when the ADS command comes back without any error but
				the compensation does not start anyway, we assume that  
				a very short compensation already has been executed. 
			*)
			Done := TRUE; (* after short timeout *)
			iState := STATE_INITIALIZATION;
		END_IF;
	END_IF

(* compensation not necessarily finished if axis stops (new modes available) - 2009-08-13 KSt *)
(*	IF NOT F_AxisHasJob(Axis.NcToPlc.StateDWord) THEN
		/* command aborted, move has been stopped before superposition finished (KSt, 12.01.2004) */
		CommandAborted := TRUE;
		iState := STATE_INITIALIZATION;
	END_IF
*)

STATE_WAITING : (* 2009-10-06 KSt  - state added for axes coupled to actual position (encoder axes or disabled axes) *)
	(* decide if superposition was completed or aborted in case of axes coupled to actual position (encoder axes or disabled axes) *)
	IF NOT F_AxisIsMoving(Axis.NcToPlc.StateDWord) THEN (* 2009-10-06 KSt *)
		(* command aborted, motion ended before superposition was finished because the axis is not moving any longer *)
		CommandAborted := TRUE;
	ELSE
		(* the initial HasJob or Moving state was the same as at end of compensation - assume that superposition completed *)
		Done := TRUE;
	END_IF
	CompensationStarted := FALSE;
	iState := STATE_INITIALIZATION;

ELSE  (* CASE : Unknown program state *)
	Error := TRUE;
	ErrorID := 16#FFFFFFFF;
	iState:= STATE_INITIALIZATION;
END_CASE

ADSbusy := fbAdsReadWrite.BUSY;
IF iState=STATE_INITIALIZATION THEN
	(* reset Busy immediately  when sequence ends *)
	IF Busy THEN
		LastExecutionResult.Done := Done;
		LastExecutionResult.CommandAborted := CommandAborted;
		LastExecutionResult.Error := Error;
		LastExecutionResult.ErrorID := ErrorID;
	END_IF
	Busy := FALSE;
	Active := FALSE;
END_IF
END_FUNCTION_BLOCK

(* POU MC_OverrideFilter, ST *)
FUNCTION_BLOCK MC_OverrideFilter
VAR_INPUT
	(* variables *)
	OverrideValueRaw		: DINT;
	(* parameter *)
	LowerOverrideThreshold	: DINT	:= 0;			(* 0...32767 digits *)
	UpperOverrideThreshold	: DINT	:= 32767;		(* 0...32767 digits *)
	OverrideSteps			: UDINT	:= 200;		(* 200 steps => 0.5 percent *)
	OverrideRecoveryTime	: TIME	:= T#150ms;	(* 150 ms *)
END_VAR
VAR_OUTPUT
	OverrideValueFiltered		: DWORD;			(* 0...1000000 counts *)
	OverridePercentFiltered	: LREAL;				(* 0...100 % *)
	Error					: BOOL;
	ErrorID					: UDINT;
END_VAR
VAR
	bFirstCycle				: BOOL := TRUE;
	bThresholdActive			: BOOL := TRUE;
	InternalOverrideValueRaw	: DINT;
	LastOverrideValueRaw		: DINT := 16#FFFF;
	OverrideRange			: DINT;
END_VAR
{library private}
VAR
	fbTimer					: TON;
END_VAR
(* default value *)
Error	:= FALSE;
ErrorID	:= MC_ERROR_NO_ERROR;

(* check parameter / error handling:   'UpperOverrideThreshold > LowerOverrideThreshold'  AND  'OverrideSteps > 1'  *)
IF( (LowerOverrideThreshold >= UpperOverrideThreshold) OR (OverrideSteps <= 1) )THEN
	OverrideValueFiltered		:= 0;
	OverridePercentFiltered	:= 0.0;
	Error	:= TRUE;
	ErrorID	:= MC_ERROR_PARAMETER_NOT_CORRECT;
	RETURN;
END_IF;

(* first cycle: timer must be elapsed *)
IF ( bFirstCycle ) THEN
	fbTimer( IN:=TRUE, PT:= T#0s );
	bFirstCycle := FALSE;
END_IF;

IF ( OverrideValueRaw >= UpperOverrideThreshold ) THEN
	InternalOverrideValueRaw := UpperOverrideThreshold;
	bThresholdActive := TRUE;
ELSIF ( OverrideValueRaw <= LowerOverrideThreshold ) THEN
	InternalOverrideValueRaw := LowerOverrideThreshold;
	bThresholdActive := TRUE;
ELSE
	InternalOverrideValueRaw := OverrideValueRaw;
	bThresholdActive := FALSE;
END_IF;

fbTimer( IN:=TRUE, PT:= OverrideRecoveryTime );
IF( fbTimer.Q = TRUE OR bThresholdActive )THEN
	OverrideRange := UpperOverrideThreshold - LowerOverrideThreshold;
(*	IF (  bThresholdActive OR ABS( InternalRawOverrideValue - LastRawOverrideValue ) >= (0.5 * OverrideRange / OverrideSteps)  ) THEN *)
(*	IF (  bThresholdActive OR ABS( InternalOverrideValueRaw - LastOverrideValueRaw ) >= ( OverrideRange / OverrideSteps)  ) THEN*)
	IF (  bThresholdActive OR ABS( InternalOverrideValueRaw - LastOverrideValueRaw ) >= ( OverrideRange / UDINT_TO_DINT(OverrideSteps))  ) THEN (* 20110511 KSt type conversion for TC3 *)
		OverrideValueFiltered := DINT_TO_DWORD(((InternalOverrideValueRaw - LowerOverrideThreshold) * 1000 / OverrideRange) * 1000);
		OverridePercentFiltered := DWORD_TO_LREAL( OverrideValueFiltered ) * LREAL#0.0001;
		LastOverrideValueRaw := InternalOverrideValueRaw;
		fbTimer( IN:=FALSE, PT:= OverrideRecoveryTime );
	END_IF;
END_IF;
END_FUNCTION_BLOCK

(* POU MC_Power, ST *)
FUNCTION_BLOCK MC_Power
(*
	Function block defined by PLCopen Part 1 - Function blocks for motion control

	This Function Block controls the power stage (on or off).

	Only 1 FB MC_Power should be issued per axis.
*)
VAR_IN_OUT
	Axis				:	AXIS_REF;	(* B *)
END_VAR
VAR_INPUT
	Enable			:	BOOL;	(* B *)
	Enable_Positive	:	BOOL;	(* E *)
	Enable_Negative	:	BOOL;	(* E *)
	Override			:	LREAL	(* V *) 	:= 100.0; (* in percent - Beckhoff proprietary input *)
	BufferMode		:	MC_BufferMode;	(* V *)
END_VAR
VAR_OUTPUT
	Status			:	BOOL;	(* B *)
	Busy			: 	BOOL;	(* V *)
	Active			: 	BOOL;	(* V *)
(*	Valid			: 	BOOL;*)	(* E *)	(* not implemented - use Busy *)
	Error			:	BOOL;	(* B *)
	ErrorID			:	UDINT;	(* E *)
END_VAR
{library private}
VAR
	EnableTimeout: TON;
	EnableOffOnDelay: TP;
(*	iOverride: DINT;*)
	iOverride: DWORD;	(* 20110511 KSt type adaption for TC3 *)
END_VAR
(*
	PlcOpen comment zu MC_Power:
		Eingänge >Override< und >BufferMode< sind Beckhoff-spezifisch 
		Ausgänge >Busy< und >Active< sind Beckhoff-spezifisch 
		Ausgang >Valid< fehlt, Funktion entspricht Active 
*)

(*EnableTimeout(IN:=Enable, PT:=T#10s);*)	(* timout if axis doesn't get ready after Enable *)
(*EnableTimeout(IN:=Enable AND NOT Status AND Axis.NcToPlc.CoupleState=0, PT:=T#10s);*) (* 2012-08-23 KSt *)	(* timout if axis doesn't get ready after Enable - just for single axes - KSt 2010-03-11 *)
EnableTimeout(IN:=Enable AND NOT Status AND Axis.NcToPlc.CoupleState=0 AND Axis.NcToPlc.ErrorCode=0, PT:=T#10s);	(* 2012-08-23 KSt *) (* timout if axis doesn't get ready after Enable - just for single axes and only if error free - KSt 2012-08-23 *)
EnableOffOnDelay(IN:= NOT Enable );	(* minimum delay between disable end re-Enable -  don't initialize before first enable *)

IF Enable THEN
	Busy := TRUE;
	Status := FALSE;
	ErrorID := 0;
	Error := FALSE;
	EnableOffOnDelay.PT:=T#50ms;	(* initialize not before first enable *)

	(* set override *)
	iOverride := LREAL_TO_DWORD(Override*10000);
	(* double check override with real and integer number because conversion may fail *)
	IF (Override < -1) OR (Override > 101) THEN	(* check real number with tolerance *)
		ErrorID := MC_ERROR_PARAMETER_NOT_CORRECT;
		Error := TRUE;
	ELSIF (iOverride < 0) OR (iOverride > 1000000) THEN	(* check integer number without tolerance *)
		ErrorID := MC_ERROR_PARAMETER_NOT_CORRECT;
		Error := TRUE;
	ELSE
		Axis.PlcToNc.Override := iOverride;
	END_IF;

	(* set enabling flags *)
	Axis.PlcToNc.ControlDWord.0 := Enable;
	Axis.PlcToNc.ControlDWord.1 := Enable_Positive;
	Axis.PlcToNc.ControlDWord.2 := Enable_Negative;

	(* set status bit *)
	(* IF  F_AxisIsReady(StateDWord := Axis.NcToPlc.StateDWord) THEN *) (* Axis ready*) 	(* 2008-12-18 KSt *)
	IF  F_AxisControlLoopClosed(StateDWord := Axis.NcToPlc.StateDWord) THEN (* Axis ready*) 	(* 2008-12-18 KSt *)
		(* status is TRUE if no error and a minimum of EnableOffOnDelay.PT (50 ms) after last recent disable *)
(*		Status := NOT Error AND NOT EnableOffOnDelay.Q; *)(* exclusive outputs *)

		(* 20101122 KSt - If control loop is closed after an error, the error is reset and the axis status is enabled *)
		(* status is TRUE after a minimum EnableOffOnDelay.PT (50 ms) after last recent disable *)
		Status := NOT EnableOffOnDelay.Q;
		IF Status THEN (* exclusive outputs *)
			Error := FALSE;
			ErrorID := 0;
		END_IF
(*	ELSIF Axis.Status.ErrorID <> 0 THEN *)(* 2009-01-29 KSt *)
	ELSIF Axis.NcToPlc.ErrorCode <> 0 THEN (* 2012-08-23 KSt *)
		Status := FALSE;
		Error := TRUE;
		(* ErrorID := Axis.Status.ErrorID;*)	(* 2015-05-05 KSt *)
		ErrorID := Axis.NcToPlc.ErrorCode;	(* 2015-05-05 KSt *)
	ELSIF EnableTimeout.Q THEN
		(* timeout after enable *)
		Status := FALSE;
		Error := TRUE;
		ErrorID := MC_ERROR_AXIS_IS_NOT_READY;
	END_IF;

ELSE (* NOT Enable *)
	(* if BufferMode=Buffered wait for current command beeing finished *)
	IF BufferMode = MC_Aborting OR NOT F_AxisHasJob(Axis.NcToPlc.StateDWord) THEN
(* changed 20100416 KSt *) (*
		Axis.PlcToNc.ControlDWord:= CLEARBIT32(Axis.PlcToNc.ControlDWord,0);
		Axis.PlcToNc.ControlDWord:= CLEARBIT32(Axis.PlcToNc.ControlDWord,1);
		Axis.PlcToNc.ControlDWord:= CLEARBIT32(Axis.PlcToNc.ControlDWord,2);	*)
		Axis.PlcToNc.ControlDWord.0 := FALSE;
		Axis.PlcToNc.ControlDWord.1 := FALSE;
		Axis.PlcToNc.ControlDWord.2:= FALSE;
		(* Override  0 % *)
		Axis.PlcToNc.Override := 0;
		Status := FALSE;
		Busy := FALSE;
		Error := FALSE;			(* reset at falling edge of Execute *)
		ErrorID := 0;
	END_IF
END_IF;

Active:=TRUE;
END_FUNCTION_BLOCK

(* POU MC_PowerStepper, ST *)
FUNCTION_BLOCK MC_PowerStepper
VAR_IN_OUT
	Axis		:	AXIS_REF;
END_VAR
VAR_INPUT
	Enable			:	BOOL;
	Enable_Positive	:	BOOL;
	Enable_Negative	:	BOOL;
	Override			:	LREAL := 100.0; (* in percent *)
	DestallParams	:	ST_PowerStepperStruct;
	KL_Status		:	USINT;
	KL_Status2		:	UINT;
END_VAR
VAR_OUTPUT
	Status			:	BOOL;
	Error			:	BOOL;
	ErrorID			:	UDINT;
	Stalled			:	BOOL;
	StallError			:	BOOL;
END_VAR
VAR
	fbPower			:	MC_Power;
	ErrorCode		:	DWORD;
	fbWriteErrCode	:	ADSWRITE;
	nRefState		:	DWORD;
	fbWriteNonRef	:	ADSWRITE;
	fbReadParams	:	ADSREAD;
	fbWriteInstOvr		:	ADSWRITE;
	bAdsInitDone		:	BOOL;

	bOverTemp		:	BOOL;
	rtOverTemp		:	R_TRIG;
	bUnderVoltage	:	BOOL;
	rtUnderVoltage	:	R_TRIG;
	bOpenLoopA		:	BOOL;
	rtOpenLoopA		:	R_TRIG;
	bOpenLoopB		:	BOOL;
	rtOpenLoopB		:	R_TRIG;
	bOverCurrentA	:	BOOL;
	rtOverCurrentA	:	R_TRIG;
	bOverCurrentB	:	BOOL;
	rtOverCurrentB	:	R_TRIG;
	rtStallError		:	R_TRIG;
	bOldState		:	BOOL;

	bLagFilterInit		: 	BOOL;
	tonLagFilter		:	TON;
	tonNoLagFilter	:	TON;

	wState2			:	WORD;
	nAngle			:	INT;
	nOldAngle		:	INT;
	AngleDiff			:	INT;
	bInErrorState		:	BOOL;

	nParamIdx		:	INT;
	bParamEnabled	:	BOOL;
	fLagLimit			:	LREAL;
	fLagFilter			:	LREAL;
	nTries			:	INT;
	tTimeOut			:	TON;
END_VAR
(*
	Aufruf des Standard-Bausteins
*)
fbPower(
	Enable:=Enable,
	Enable_Positive:=Enable_Positive,
	Enable_Negative:=Enable_Negative,
	Override:=Override,
	Axis:=Axis);

(*
	Ein paar Vorbereitungen ...
*)
wState2:=UINT_TO_WORD(KL_Status2);
bInErrorState:=Axis.NcToPlc.ErrorCode<>0;
nAngle:=SHR(USINT_TO_BYTE(KL_Status),1) AND 7;
AngleDiff:=nAngle-nOldAngle;
nOldAngle:=nAngle;
IF((Axis.NcToPlc.StateDWord AND 16#0000001C)=16#0000001C)THEN		(* Ziel erreicht *)
	nTries:=0;
END_IF
IF((Axis.NcToPlc.StateDWord AND 16#00000080)=16#00000080)THEN		(* Stop *)
	nTries:=0;
END_IF

(* ======================================
	Parameter-Lademaschine
====================================== *)
IF(NOT Enable)THEN
	(*
		Reinitialisieren
	*)
	nParamIdx:=0;
	bParamEnabled:=FALSE;
	fbReadParams(
		NETID:='', PORT:=AMSPORT_R0_NCSAF, IDXGRP:=0, IDXOFFS:=0,
		LEN:=0, DESTADDR:=0,
		READ:=FALSE, TMOUT:=T#5s);
ELSE
	IF(NOT bParamEnabled)THEN
		CASE nParamIdx OF
			0:
				IF(NOT fbReadParams.READ)THEN
					fbReadParams.LEN:=SIZEOF(fLagLimit);
					fbReadParams.DESTADDR:=ADR(fLagLimit);
					fbReadParams.IDXGRP:=16#00004000+Axis.NcToPlc.AxisId;
					fbReadParams.IDXOFFS:=16#00020012;
					fbReadParams.READ:=TRUE;
				ELSIF(NOT fbReadParams.BUSY)THEN
					IF(fbReadParams.ERR)THEN
						fLagLimit:=5.0;
					END_IF
					fbReadParams.READ:=FALSE;
					nParamIdx:=nParamIdx+1;
				END_IF
				fbReadParams(NETID:='', PORT:=AMSPORT_R0_NCSAF, TMOUT:=T#5s);
			1:
				IF(NOT fbReadParams.READ)THEN
					fbReadParams.LEN:=SIZEOF(fLagFilter);
					fbReadParams.DESTADDR:=ADR(fLagFilter);
					fbReadParams.IDXGRP:=16#00004000+Axis.NcToPlc.AxisId;
					fbReadParams.IDXOFFS:=16#00020013;
					fbReadParams.READ:=TRUE;
				ELSIF(NOT fbReadParams.BUSY)THEN
					IF(fbReadParams.ERR)THEN
						fLagFilter:=0.1;
					END_IF
					fbReadParams.READ:=FALSE;
					nParamIdx:=nParamIdx+1;
					tonLagFilter(IN:=FALSE, PT:=T#10ms);
					tonNoLagFilter(IN:=NOT tonLagFilter.IN, PT:=T#10ms);
				END_IF
				fbReadParams(NETID:='', PORT:=AMSPORT_R0_NCSAF, TMOUT:=T#5s);
			ELSE
				bParamEnabled:=TRUE;
		END_CASE
	END_IF
END_IF

IF(fbPower.Error)THEN
	ErrorID := fbPower.ErrorID;
	Error := TRUE;
	Status := bAdsInitDone := FALSE;
ELSIF(NOT Enable)THEN
	ErrorID := 0;
	Error := Status := bAdsInitDone := FALSE;
ELSE
	(*
		Sicherstellen, dass die ADS-FBs initialisiert sind
	*)
	IF(NOT bAdsInitDone)THEN
		bAdsInitDone := TRUE;
		fbWriteNonRef(
			WRITE:=FALSE,
			NETID:='',
			PORT:=AMSPORT_R0_NCSAF,
			IDXGRP:=16#00004200+Axis.NcToPlc.AxisId,
			IDXOFFS:=16#0000001B,
			LEN:=SIZEOF(nRefState),
			SRCADDR:=ADR(nRefState),
			TMOUT:=T#5s,
			);
		fbWriteInstOvr(
			WRITE:=FALSE,
			NETID:='',
			PORT:=AMSPORT_R0_NCSAF,
			IDXGRP:=16#00004200+Axis.NcToPlc.AxisId,
			IDXOFFS:=16#00000029,
			LEN:=0,
			SRCADDR:=0,
			TMOUT:=T#5s,
			);
		fbWriteErrCode(
			WRITE:=FALSE,
			NETID:='',
			PORT:=AMSPORT_R0_NCSAF,
			IDXGRP:=16#00004200+Axis.NcToPlc.AxisId,
			IDXOFFS:=16#00000019,
			LEN:=SIZEOF(ErrorCode),
			SRCADDR:=ADR(ErrorCode),
			TMOUT:=T#5s,
			);
	END_IF

	(*
		Zentrales Versenden für Kommandos zur instantanen Override-Änderung
		Dies muss vor der Stelle des Test liegen, damit der Override-Wert im Mapping sicher angekommen ist,
		wenn dieses Kommando per ADS eintrifft.
	*)
	fbWriteInstOvr(
		NETID:='',
		PORT:=AMSPORT_R0_NCSAF,
		IDXGRP:=16#00004200+Axis.NcToPlc.AxisId,
		IDXOFFS:=16#00000029,
		LEN:=0,
		SRCADDR:=0,
		TMOUT:=T#5s,
		);
	IF(NOT fbWriteInstOvr.BUSY)THEN
		fbWriteInstOvr.WRITE:=FALSE;
	END_IF

	bLagFilterInit:=bLagFilterInit OR tonLagFilter.Q;

	IF(DestallParams.DestallEnable)THEN
		(*
			Stall Detection
		*)
		bOldState:=Stalled;
		CASE DestallParams.DestallDetectMode OF
			PwStDetectMode_Encoderless:
				Stalled:=ABS(AngleDiff)>=4;
			PwStDetectMode_Lagging:
				IF(bParamEnabled)THEN
					IF(fLagFilter<=0.001)THEN
						tonLagFilter(IN:=FALSE, PT:=T#10ms);
						tonNoLagFilter(IN:=NOT tonLagFilter.IN, PT:=T#10ms);
						Stalled:=ABS(Axis.NcToPlc.PosDiff)>=fLagLimit;
					ELSE
						tonLagFilter(IN:=(ABS(Axis.NcToPlc.PosDiff)>=fLagLimit), PT:=LREAL_TO_TIME(fLagFilter*1000.0));
						tonNoLagFilter(IN:=NOT tonLagFilter.IN, PT:=LREAL_TO_TIME(fLagFilter*1000.0));
						Stalled:=tonLagFilter.Q;
					END_IF
				ELSE
					tonLagFilter(IN:=FALSE, PT:=T#10ms);
					tonNoLagFilter(IN:=NOT tonLagFilter.IN, PT:=T#10ms);
					Stalled:=FALSE;
				END_IF
			ELSE
				Stalled:=FALSE;
		END_CASE
		IF(NOT bOldState AND Stalled)THEN
			nTries:=nTries+1;
		END_IF
		(*
			Stall Handling
		*)
		StallError:=StallError AND (bInErrorState  OR fbWriteErrCode.WRITE);
		bOldState:=StallError;
		CASE DestallParams.DestallMode OF
			PwStMode_None:
				StallError:=FALSE;
				tTimeOut(IN:=FALSE, PT:=T#10ms);
			PwStMode_SetError:
				StallError:=StallError OR Stalled;
				tTimeOut(IN:=FALSE, PT:=T#10ms);
			PwStMode_SetErrNonRef:
				StallError:=StallError OR Stalled;
				IF(Stalled AND ((Axis.NcToPlc.StateDWord AND 16#00000002)<>0) )THEN
					nRefState:=0;
					fbWriteNonRef.WRITE:=TRUE;
				END_IF
				tTimeOut(IN:=FALSE, PT:=T#10ms);
			PwStMode_UseOverride:
				IF(Stalled OR (bLagFilterInit AND NOT tonNoLagFilter.Q))THEN	(* HKP *)
					Axis.PlcToNc.Override := 0;
					fbWriteInstOvr.WRITE:=TRUE;
				END_IF
				tTimeOut(IN:=Stalled, PT:=MAX(DestallParams.Timeout, T#10ms));
				StallError:=StallError OR tTimeOut.Q;
				IF(nTries>DestallParams.Retries)THEN
					StallError:=TRUE;
				END_IF
		END_CASE

		IF(StallError AND NOT bOldState)THEN
			ADSLOGDINT((ADSLOG_MSGTYPE_ERROR OR ADSLOG_MSGTYPE_LOG), 'MC_PowerStepper (AxisID: %d) reporting error 0x4636 (stall error) !', DWORD_TO_DINT(Axis.NcToPlc.AxisId));
		END_IF
		rtStallError(CLK:=StallError AND NOT bInErrorState AND NOT fbWriteErrCode.WRITE);
		IF(rtStallError.Q)THEN
			ErrorCode:=16#00004636;
			fbWriteErrCode.WRITE:=TRUE;
		END_IF

	END_IF

	Status:=TRUE;
	IF(DestallParams.StatusMonEnable)THEN
		(*
			State Monitoring
		*)
		bOldState:=bOverTemp;
		bOverTemp:=(wState2 AND 2#0000000100000000)<>0;
		Status:=Status AND NOT bOverTemp;
		IF(bOverTemp AND NOT bOldState)THEN
			ADSLOGDINT((ADSLOG_MSGTYPE_ERROR OR ADSLOG_MSGTYPE_LOG), 'MC_PowerStepper (AxisID: %d) reporting error 0x4630 (overtemperature, KL terminal) !', DWORD_TO_DINT(Axis.NcToPlc.AxisId));
		END_IF
		rtOverTemp(CLK:=bOverTemp AND NOT bInErrorState AND NOT fbWriteErrCode.WRITE);
		IF(rtOverTemp.Q)THEN
			ErrorCode:=16#00004630;
			fbWriteErrCode.WRITE:=TRUE;
		END_IF
		bOverTemp:=bOverTemp AND (bInErrorState  OR fbWriteErrCode.WRITE);
		bOldState:=bUnderVoltage;
		bUnderVoltage:=(wState2 AND 2#0000001000000000)<>0;
		Status:=Status AND NOT bUnderVoltage;
		IF(bUnderVoltage AND NOT bOldState)THEN
						ADSLOGDINT((ADSLOG_MSGTYPE_ERROR OR ADSLOG_MSGTYPE_LOG), 'MC_PowerStepper (AxisID: %d) reporting error 0x4631 (bad supply voltage, KL terminal) !', DWORD_TO_DINT(Axis.NcToPlc.AxisId));
		END_IF
		rtUnderVoltage(CLK:=bUnderVoltage AND NOT bInErrorState AND NOT fbWriteErrCode.WRITE);
		IF(rtUnderVoltage.Q)THEN
			ErrorCode:=16#00004631;
			fbWriteErrCode.WRITE:=TRUE;
		END_IF
		bUnderVoltage:=bUnderVoltage AND (bInErrorState  OR fbWriteErrCode.WRITE);
		bOldState:=bOpenLoopA;
		bOpenLoopA:=(wState2 AND 2#0000010000000000)<>0;
		Status:=Status AND NOT bOpenLoopA;
		IF(bOpenLoopA AND NOT bOldState)THEN
			ADSLOGDINT((ADSLOG_MSGTYPE_ERROR OR ADSLOG_MSGTYPE_LOG), 'MC_PowerStepper (AxisID: %d) reporting error 0x4632 (open loop, phase A) !', DWORD_TO_DINT(Axis.NcToPlc.AxisId));
		END_IF
		rtOpenLoopA(CLK:=bOpenLoopA AND NOT bInErrorState AND NOT fbWriteErrCode.WRITE);
		IF(rtOpenLoopA.Q)THEN
			ErrorCode:=16#00004632;
			fbWriteErrCode.WRITE:=TRUE;
		END_IF
		bOpenLoopA:=bOpenLoopA AND (bInErrorState  OR fbWriteErrCode.WRITE);
		bOldState:=bOpenLoopB;
		bOpenLoopB:=(wState2 AND 2#0000100000000000)<>0;
		Status:=Status AND NOT bOpenLoopB;
		IF(bOpenLoopB AND NOT bOldState)THEN
			ADSLOGDINT((ADSLOG_MSGTYPE_ERROR OR ADSLOG_MSGTYPE_LOG), 'MC_PowerStepper (AxisID: %d) reporting error 0x4633 (open loop, phase B) !', DWORD_TO_DINT(Axis.NcToPlc.AxisId));
		END_IF
		rtOpenLoopB(CLK:=bOpenLoopB AND NOT bInErrorState AND NOT fbWriteErrCode.WRITE);
		IF(rtOpenLoopB.Q)THEN
			ErrorCode:=16#00004633;
			fbWriteErrCode.WRITE:=TRUE;
		END_IF
		bOpenLoopB:=bOpenLoopB AND (bInErrorState  OR fbWriteErrCode.WRITE);
		bOldState:=bOverCurrentA;
		bOverCurrentA:=(wState2 AND 2#0001000000000000)<>0;
		Status:=Status AND NOT bOverCurrentA;
		IF(bOverCurrentA AND NOT bOldState)THEN
			ADSLOGDINT((ADSLOG_MSGTYPE_ERROR OR ADSLOG_MSGTYPE_LOG), 'MC_PowerStepper (AxisID: %d) reporting error 0x4634 (overcurrent, phase A) !', DWORD_TO_DINT(Axis.NcToPlc.AxisId));
		END_IF
		rtOverCurrentA(CLK:=bOverCurrentA AND NOT bInErrorState AND NOT fbWriteErrCode.WRITE);
		IF(rtOverCurrentA.Q)THEN
			ErrorCode:=16#00004634;
			fbWriteErrCode.WRITE:=TRUE;
		END_IF
		bOverCurrentA:=bOverCurrentA AND (bInErrorState  OR fbWriteErrCode.WRITE);
		bOldState:=bOverCurrentB;
		bOverCurrentB:=(wState2 AND 2#0010000000000000)<>0;
		Status:=Status AND NOT bOverCurrentB;
		IF(bOverCurrentB AND NOT bOldState)THEN
			ADSLOGDINT((ADSLOG_MSGTYPE_ERROR OR ADSLOG_MSGTYPE_LOG), 'MC_PowerStepper (AxisID: %d) reporting error 0x4635 (overcurrent, phase B) !', DWORD_TO_DINT(Axis.NcToPlc.AxisId));
		END_IF
		rtOverCurrentB(CLK:=bOverCurrentB AND NOT bInErrorState AND NOT fbWriteErrCode.WRITE);
		IF(rtOverCurrentB.Q)THEN
			ErrorCode:=16#00004635;
			fbWriteErrCode.WRITE:=TRUE;
		END_IF
		bOverCurrentB:=bOverCurrentB AND (bInErrorState  OR fbWriteErrCode.WRITE);
	END_IF

	(*
		Zentrale Versendung von Achs-ErrorCodes
	*)
	fbWriteErrCode(
		NETID:='',
		PORT:=AMSPORT_R0_NCSAF,
		IDXGRP:=16#00004200+Axis.NcToPlc.AxisId,
		IDXOFFS:=16#00000019,
		LEN:=SIZEOF(ErrorCode),
		SRCADDR:=ADR(ErrorCode),
		TMOUT:=T#5s,
		);
	IF(bInErrorState)THEN
		fbWriteErrCode.WRITE:=FALSE;
	END_IF

	(*
		Zentrale Versendung von Referenz-Resets
	*)
	fbWriteNonRef(
		NETID:='',
		PORT:=AMSPORT_R0_NCSAF,
		IDXGRP:=16#00004200+Axis.NcToPlc.AxisId,
		IDXOFFS:=16#0000001B,
		LEN:=SIZEOF(nRefState),
		SRCADDR:=ADR(nRefState),
		TMOUT:=T#5s,
		);
	IF(NOT fbWriteNonRef.BUSY)THEN
		fbWriteNonRef.WRITE:=FALSE;
	END_IF

END_IF
END_FUNCTION_BLOCK

(* POU MC_ReadActualPosition, ST *)
FUNCTION_BLOCK MC_ReadActualPosition
(*	This Function Block returns the actual position. *)
VAR_IN_OUT
	Axis			:	AXIS_REF;	(* B *)
END_VAR
VAR_INPUT
	Enable		:	BOOL;		(* B *)
END_VAR
VAR_OUTPUT
	Valid		:	BOOL;		(* B *)
	Busy		:	BOOL;		(* E *)
	Error		:	BOOL;		(* B *)
	ErrorID		:	UDINT;		(* E *)
	Position		:	LREAL;		(* B *)
END_VAR
VAR
END_VAR
Error := FALSE;
ErrorID := 0;
IF Enable THEN
	Busy := TRUE;
	Position := Axis.NcToPlc.ActPos;
	Valid := TRUE;
ELSE
	Busy := FALSE;
	Position := 0.0;
	Valid := FALSE;
END_IF;
END_FUNCTION_BLOCK

(* POU MC_ReadActualVelocity, ST *)
FUNCTION_BLOCK MC_ReadActualVelocity
(*
	This Function Block returns the value of the actual velocity as long as Enable is 
	set. Valid is true when the data-output ActualVelocity is valid. If Enable is reset, the 
	data loses its validity, and all outputs are reset, no matter if new data is available.
*)
VAR_IN_OUT
	Axis			:	AXIS_REF;	(* B *)
END_VAR
VAR_INPUT
	Enable 		: 	BOOL;	(* B *)
END_VAR
VAR_OUTPUT
	Valid 		: 	BOOL;	(* B *)
	Busy 		: 	BOOL;	(* E *)
	Error 		: 	BOOL;	(* B *)
	ErrorID 		: 	UDINT;	(* E *)
	ActualVelocity (* Velocity *): 	LREAL;	(* B *)
END_VAR
VAR
END_VAR
Error := FALSE;
ErrorID := 0;
IF Enable THEN
	Busy := TRUE;
	Valid := TRUE;
	ActualVelocity := Axis.NcToPlc.ActVelo;
ELSE
	Busy := FALSE;
	Valid := FALSE;
	ActualVelocity := 0;
END_IF
END_FUNCTION_BLOCK

(* POU MC_ReadApplicationRequest, ST *)
FUNCTION_BLOCK MC_ReadApplicationRequest
(*	This Function Block returns a data set containing all parameters of an application request *)
VAR_IN_OUT
	ApplicationRequest 	: 	ST_NcApplicationRequest;
	Axis			:	AXIS_REF;
END_VAR
VAR_INPUT
	Execute		: 	BOOL;
END_VAR
VAR_OUTPUT
	Done 		: 	BOOL;
	Busy		: 	BOOL;
	Error 		: 	BOOL;
	ErrorID 		: 	UDINT;
	Request		: 	BOOL;		(* application request bit [0/1] *)
	RequestType	: 	UINT;		(* application request TYPE/ID *)
END_VAR
VAR
	TriggerExecute: R_TRIG;
	state: _E_TcMC_STATES := STATE_INITIALIZATION;
	fbAdsRead		: 	ADSREAD;
END_VAR
TriggerExecute(CLK:=Execute);

CASE state OF
	STATE_INITIALIZATION:
		IF NOT Execute THEN
			Done := FALSE;
			Error := FALSE;	(* reset at falling edge of Execute *)
			ErrorID := 0;
		END_IF
		IF TriggerExecute.Q THEN
			Done := FALSE;
			Busy := TRUE;
			Error := FALSE;
			ErrorID := 0;
			Request := FALSE;
			RequestType := 0 ;
			fbAdsRead(READ:=FALSE);
		END_IF
		IF Busy THEN
			fbAdsRead(
				NETID:= TcMcGlobal.NCNETID_TCMC,
				PORT:= TcMcGlobal.NCPORT_TCMC,
				IDXGRP:=TcMcGlobal.Axis.Parameter.IDXGRP+Axis.NcToPlc.AxisId,
				IDXOFFS:= TcMcGlobal.Axis.Parameter.IDXOFFS.APPLICATIONREQUEST,
				LEN:= SIZEOF(ApplicationRequest),
				DESTADDR:= ADR(ApplicationRequest),
				READ:= TRUE,
				TMOUT:= TcMcGlobal.tADSTimeOut );
			IF NOT fbAdsRead.BUSY THEN
				Error := fbAdsRead.ERR;
				ErrorID := fbAdsRead.ERRID;
				Done := NOT Error;
				IF Done THEN
					Request := ApplicationRequest.bApplRequestBit<>0;
					RequestType := ApplicationRequest.nApplRequestType;
				END_IF
				Busy := FALSE;
			END_IF
		END_IF
END_CASE
END_FUNCTION_BLOCK

(* POU MC_ReadAxisComponents, ST *)
FUNCTION_BLOCK  MC_ReadAxisComponents
VAR_IN_OUT
	AxisComponents 	: 	ST_AxisComponents;
	Axis				:	AXIS_REF;
END_VAR
VAR_INPUT
	Execute: BOOL;
END_VAR
VAR_OUTPUT
	Done : BOOL;
	Busy: BOOL;
	Error : BOOL;
	ErrorID : UDINT;
END_VAR
VAR
	TriggerExecute: R_TRIG;
	state: _E_TcMC_STATES := STATE_INITIALIZATION;
	fbAdsRead		: 	ADSREAD;
END_VAR
TriggerExecute(CLK:=Execute);

CASE state OF
	STATE_INITIALIZATION:
		IF NOT Execute THEN
			Done := FALSE;
			Error := FALSE;	(* reset at falling edge of Execute *)
			ErrorID := 0;
		END_IF
		IF TriggerExecute.Q THEN
			Done := FALSE;
			Busy := TRUE;
			Error := FALSE;
			ErrorID := 0;
			fbAdsRead(READ:=FALSE);
		END_IF
		IF Busy THEN
			fbAdsRead(
				NETID:= TcMcGlobal.NCNETID_TCMC,
				PORT:= TcMcGlobal.NCPORT_TCMC,
				IDXGRP:=TcMcGlobal.Axis.Parameter.IDXGRP+Axis.NcToPlc.AxisId,
				IDXOFFS:= 16#5A,
				LEN:= SIZEOF(AxisComponents),
				DESTADDR:= ADR(AxisComponents),
				READ:= TRUE,
				TMOUT:= TcMcGlobal.tADSTimeOut );
			IF NOT fbAdsRead.BUSY THEN
				Error := fbAdsRead.ERR;
				ErrorID := fbAdsRead.ERRID;
				Done := NOT Error;
				Busy := FALSE;
			END_IF
		END_IF
END_CASE
END_FUNCTION_BLOCK

(* POU MC_ReadAxisError, ST *)
FUNCTION_BLOCK MC_ReadAxisError
(*
	This Function Block presents general axis errors not relating to the Function Blocks. 
	(for instance axis errors, drive errors, communication errors)
 *)
VAR_IN_OUT
	Axis				:	AXIS_REF;	(* B *)
END_VAR
VAR_INPUT
	Enable			:	BOOL;		(* B *)
END_VAR
VAR_OUTPUT
	Valid			:	BOOL;		(* B *)
	Busy			:	BOOL;		(* E *)
	Error			:	BOOL;		(* B *)
	ErrorID			:	DWORD;	(* B *)
	AxisErrorID		:	DWORD;	(* B *)
END_VAR
VAR
END_VAR
IF Enable THEN
	Busy		 := TRUE;
	Valid 		:=  TRUE;
	ErrorID 		:= 0;
	AxisErrorID 	:= Axis.NcToPlc.ErrorCode;
	Error		:= ErrorID <> 0;
ELSE
	Busy 		:= FALSE;
	Valid 		:= FALSE;
	Error 		:= FALSE;	(* reset at falling edge of Execute *)
	ErrorID 		:= 0;
	AxisErrorID 	:= 0;
END_IF;
END_FUNCTION_BLOCK

(* POU MC_ReadBoolParameter, ST *)
FUNCTION_BLOCK MC_ReadBoolParameter
(*	This Function Block returns the value of a vendor specific boolean parameter.*)
VAR_IN_OUT
	Axis					:	AXIS_REF;	(* B *)
END_VAR
VAR_INPUT
	Enable				:	BOOL;		(* B *)
	ParameterNumber		:	INT;			(* B *)
	ReadMode			:	E_ReadMode(* V *)	:= ReadMode_Once;	 (* Beckhoff proprietary input *)
END_VAR
VAR_OUTPUT
	Valid				:	BOOL;	(* B *)
	Busy				: 	BOOL;	(* E *)
	Error				:	BOOL;	(* B *)
	ErrorID				:	UDINT;	(* E *)
	Value				:	BOOL;	(* B *)
END_VAR
VAR
	ADSbusy: BOOL;
	fbReadWriteParameter: 	_FB_ReadWriteParameter;
END_VAR
{library private}
VAR
	nParatype 			: 	_E_ParameterType;
	dwValue 				: 	DWORD;
	lrValue				: 	LREAL;
	bStarted				:	BOOL;
	fbTrigger 			: 	R_TRIG;
END_VAR
IF NOT Enable THEN
	Valid := FALSE;
	Error := FALSE;			(* reset at falling edge of Execute *)
	ErrorID := 0;
END_IF
IF ReadMode = ReadMode_Once THEN
	fbTrigger(CLK:= Enable);
	IF fbTrigger.Q AND NOT bStarted THEN
		bStarted := TRUE;
		Valid := FALSE;
		Error := FALSE;
		ErrorID := MC_ERROR_NO_ERROR;
	END_IF;
ELSE
	IF Enable AND NOT bStarted THEN
		bStarted := TRUE;
		Valid := FALSE;
		Error := FALSE;
		ErrorID := MC_ERROR_NO_ERROR;
	END_IF;
END_IF;
(* *)
IF bStarted THEN
	nParatype := PARAMETERTYPE_BOOL;
	fbReadWriteParameter(Enable:= TRUE, ParameterNumber:= ParameterNumber, Mode:= READWRITEPARAMETERMODE_READ,
						ParameterType:=nParatype, Axis:= Axis, ValueLreal:= lrValue, ValueDword := dwValue, ValueBool := Value);
	IF fbReadWriteParameter.Done THEN
		bStarted := FALSE;
		Valid := TRUE;
		fbReadWriteParameter(Enable:= FALSE, ParameterNumber:= ParameterNumber, Mode:= READWRITEPARAMETERMODE_READ,
						ParameterType:= nParatype , Axis:= Axis, ValueLreal:= lrValue, ValueDword := dwValue, ValueBool := Value);
	END_IF;
	IF fbReadWriteParameter.Error THEN
		bStarted := FALSE;
		Valid := FALSE;
		Error := TRUE;
		ErrorID := fbReadWriteParameter.ErrorID;
		fbReadWriteParameter(Enable:= FALSE, ParameterNumber:= ParameterNumber, Mode:= READWRITEPARAMETERMODE_READ,
						ParameterType:= nParatype , Axis:= Axis, ValueLreal:= lrValue, ValueDword := dwValue, ValueBool := Value);
	END_IF;
END_IF;

ADSbusy := fbReadWriteParameter.ADSbusy;
Busy := (Enable AND ReadMode<>ReadMode_Once) OR bStarted;
END_FUNCTION_BLOCK

(* POU MC_ReadDriveAddress, ST *)
FUNCTION_BLOCK MC_ReadDriveAddress
(*	This Function Block returns the value of a vendor specific parameter *)
VAR_IN_OUT
	Axis				: AXIS_REF;	(* B *)
END_VAR
VAR_INPUT
	Execute			: BOOL;
END_VAR
VAR_OUTPUT
	Done 			: BOOL;
	Busy			: BOOL;
	Error			: BOOL;
	ErrorID			: UDINT;
	DriveAddress 	: ST_DriveAddress;
END_VAR
VAR
	state			: 	_E_TcMC_STATES := STATE_INITIALIZATION;
	TriggerExecute: R_TRIG;
	fbAdsRead: ADSREAD;
	readBuffer			: ARRAY[0..63] OF BYTE;	(* 2013-04-03 KSt - new data structure - size changed from 10 to 64 bytes *)
END_VAR
{ library private }
VAR
	i: INT;
	pDword : POINTER TO DWORD;
END_VAR
TriggerExecute(CLK:=Execute);

CASE state OF
	STATE_INITIALIZATION:
		IF NOT Execute THEN
			Done := FALSE;
			Error := FALSE;	(* reset at falling edge of Execute *)
			ErrorID := 0;
		END_IF
		IF TriggerExecute.Q THEN
			Done := FALSE;
			Busy := TRUE;
			Error := FALSE;
			ErrorID := 0;
			fbAdsRead(READ:=FALSE);
			(* read version of NC - 2013-04-03 KSt - read version dependent structure size *)
			IF TcMcGlobal.NcDeviceInfoNcVersion=0 THEN
				TcMcGlobal.ReadDeviceInfo();
				state := STATE_WAITING;
			ELSE
				state := STATE_ORDER;
			END_IF
		END_IF

	STATE_WAITING : (* 2013-09-04 - new waiting state in case of invalid NC version information *)
		(* check for NC version *)
		TcMcGlobal.ReadDeviceInfo();
		IF NOT TcMcGlobal.fbADSRDDEVINFO.BUSY THEN
			state := STATE_ORDER;
		END_IF

	STATE_ORDER :
			IF TcMcGlobal.NcDeviceInfoNcVersion >= 16#03010FA2 (* Tc 3.1 NC4002 *) THEN
				fbAdsRead.LEN := SIZEOF(readBuffer);
			ELSIF TcMcGlobal.NcDeviceInfoNcVersion<16#03010000 AND TcMcGlobal.NcDeviceInfoNcVersion >= 16#03000BDB (* Tc 3.0 NC3035 *) THEN
				fbAdsRead.LEN := SIZEOF(readBuffer);
			ELSIF TcMcGlobal.NcDeviceInfoNcVersion<16#03000000 AND TcMcGlobal.NcDeviceInfoNcVersion >= 16#020B08B7 (* Tc 2.11 NC2231 *) THEN
				fbAdsRead.LEN := SIZEOF(readBuffer);
			ELSE
				MEMSET(ADR(readBuffer), SIZEOF(readBuffer), 0);
				fbAdsRead.LEN :=10; (* use old readbuffer size for compatibility reasons *)
			END_IF
			fbAdsRead(
				NETID:= TcMcGlobal.NCNETID_TCMC,
				PORT:= TcMcGlobal.NCPORT_TCMC,
				IDXGRP:=TcMcGlobal.Axis.Parameter.IDXGRP+Axis.NcToPlc.AxisId,
				IDXOFFS:= TcMcGlobal.Axis.Parameter.IDXOFFS.HWAMSADDR,
				LEN:= (* see above *),
				DESTADDR:= ADR(readBuffer),
				READ:= TRUE,
				TMOUT:= TcMcGlobal.tADSTimeOut );
			state := STATE_RUNNING;

	STATE_RUNNING:  (* wait until command is accepted *)
		fbAdsRead();
		IF NOT fbAdsRead.BUSY THEN
			Error := fbAdsRead.ERR;
			ErrorID := fbAdsRead.ERRID;
			IF NOT Error THEN
				FOR i := 0 TO 5 DO
					DriveAddress.NetIdBytes[i] := readBuffer[i];
				END_FOR
				DriveAddress.NetID := F_CreateAmsNetId( DriveAddress.NetIdBytes );
				DriveAddress.SlaveAddress := readBuffer[6] + 256* readBuffer[7];
				DriveAddress.Channel := readBuffer[8];
				pDword := ADR(readBuffer[12]);
				DriveAddress.NcDriveId := pDword^;
				pDword := ADR(readBuffer[16]);
				DriveAddress.NcDriveIndex := pDword^;
				pDword := ADR(readBuffer[20]);
				DriveAddress.NcDriveType := pDword^;
				pDword := ADR(readBuffer[24]);
				DriveAddress.NcEncoderId := pDword^;
				pDword := ADR(readBuffer[28]);
				DriveAddress.NcEncoderIndex := pDword^;
				pDword := ADR(readBuffer[32]);
				DriveAddress.NcEncoderType := pDword^;
				pDword := ADR(readBuffer[36]);
				DriveAddress.NcAxisId := pDword^;
				pDword := ADR(readBuffer[40]);
				DriveAddress.NcAxisType := pDword^;
			END_IF
			Done := NOT Error;
			Busy := FALSE;
			fbAdsRead(READ:=FALSE);
			state := STATE_INITIALIZATION;  (* wait until command is accepted *)
		END_IF
END_CASE
END_FUNCTION_BLOCK

(* POU MC_ReadParameterSet, ST *)
FUNCTION_BLOCK  MC_ReadParameterSet
(*	This Function Block returns the complete set of axis parameters *)
VAR_IN_OUT
	Parameter 	: 	ST_AxisParameterSet;
	Axis			:	AXIS_REF;
END_VAR
VAR_INPUT
	Execute		: 	BOOL;
END_VAR
VAR_OUTPUT
	Done 		: 	BOOL;
	Busy		: 	BOOL;
	Error 		: 	BOOL;
	ErrorID 		: 	UDINT;
END_VAR
VAR
	TriggerExecute: R_TRIG;
	state: _E_TcMC_STATES := STATE_INITIALIZATION;
	fbAdsRead		: 	ADSREAD;
	SizeofPayloadData : UDINT;
END_VAR
TriggerExecute(CLK:=Execute);

CASE state OF
	STATE_INITIALIZATION:
		IF NOT Execute THEN
			Done := FALSE;
			Error := FALSE;	(* reset at falling edge of Execute *)
			ErrorID := 0;
		END_IF
		IF TriggerExecute.Q THEN
			Done := FALSE;
			Busy := TRUE;
			Error := FALSE;
			ErrorID := 0;
			fbAdsRead(READ:=FALSE);
			IF TcMcGlobal.NcDeviceInfoNcVersion=0 THEN
				TcMcGlobal.ReadDeviceInfo();
				state := STATE_WAITING;
			ELSE
				state := STATE_ORDER;
			END_IF
		END_IF

	STATE_WAITING :
		(* check for NC version *)
		TcMcGlobal.ReadDeviceInfo();
		IF TcMcGlobal.NcDeviceInfoNcVersion<>0 THEN
			state := STATE_ORDER;
		ELSIF TcMcGlobal.fbADSRDDEVINFO.ERR THEN
			Error := TRUE;
			ErrorID := TcMcGlobal.fbADSRDDEVINFO.ERRID;
			Busy := FALSE;
			state := STATE_INITIALIZATION;
		END_IF

	STATE_ORDER :
		ActGetSizeOfParameterSet();		(* 2011-06-29 KSt - get size for differently aligned systems *)
		fbAdsRead(
			NETID:= TcMcGlobal.NCNETID_TCMC,
			PORT:= TcMcGlobal.NCPORT_TCMC,
			IDXGRP:=TcMcGlobal.Axis.Parameter.IDXGRP+Axis.NcToPlc.AxisId,
			IDXOFFS:= (* 16#00 + *) Axis.NcToPlc.ControlLoopIndex * 16#00100000,
(*			LEN:= SIZEOF(Parameter),*)	(* 2011-06-29 KSt - get size for differently aligned systems *)
			LEN:= ,						(* 2011-06-29 KSt - get size for differently aligned systems *)
			DESTADDR:= ADR(Parameter),
			READ:= TRUE,
			TMOUT:= TcMcGlobal.tADSTimeOut );
		IF NOT fbAdsRead.BUSY THEN
			Error := fbAdsRead.ERR;
			ErrorID := fbAdsRead.ERRID;
			Done := NOT Error;
			Busy := FALSE;
			state := STATE_INITIALIZATION;
		END_IF

END_CASE
END_FUNCTION_BLOCK
ACTION ActGetSizeOfParameterSet:
(* adjustment of the data size to different system with different alignement *)

SizeofPayloadData := DWORD_TO_UDINT( ADR(Parameter.arrReserved) - ADR(Parameter) );

IF SIZEOF(Parameter) < (1024 + 512) / 2 THEN
	(* TC2 environment
	 	set the size of the data structure to 512 if the payload data size (data without reserved bytes) is smaller,
		Otherwise set the size to the size of the payload data.
	*)
	IF TcMcGlobal.NcDeviceInfoNcVersion >= 16#020B049C THEN	(* from 2.11 NC 1180 *)
		fbAdsRead.LEN := MAX( SizeofPayloadData, 512 );
	ELSE
		(* use 512 for any older system with smaller structure definition *)
		fbAdsRead.LEN := 512;
	END_IF
ELSE
	(* TC3 environment with extended size
		set the size of the data structure to 1024 if the payload data size (data without reserved bytes) is smaller,
		Otherwise set the size to the size of the payload data.
	*)
	fbAdsRead.LEN := MAX( SizeofPayloadData, 1024 );
END_IF
END_ACTION

(* POU MC_ReadStatus, ST *)
FUNCTION_BLOCK MC_ReadStatus
(*	This Function Block returns in detail the status of the axis with respect to the motion currently in progress *)
VAR_IN_OUT
	Axis				:	AXIS_REF;	(* B *)
END_VAR
VAR_INPUT
	Enable			:	BOOL;	(* B *)
END_VAR
VAR_OUTPUT
	Valid			:	BOOL;	(* B *)
	Busy			: 	BOOL;	(* E *)
	Error			:	BOOL;	(* B *)
	ErrorID			:	UDINT;	(* E *)
	(* motion control statemachine states: *)
	ErrorStop		:	BOOL;	(* B *)
	Disabled			:	BOOL;	(* B *)
	Stopping			:	BOOL;	(* B *)
	StandStill		:	BOOL;	(* B *)
	DiscreteMotion	:	BOOL;	(* B *)
	ContinuousMotion	:	BOOL;	(* B *)
	SynchronizedMotion:	BOOL;	(* E *)
	Homing			:	BOOL;	(* E *)
	(* additional status *)
	ConstantVelocity	:	BOOL;	(* V *)
	Accelerating		:	BOOL;	(* V *)
	Decelerating		:	BOOL;	(* V *)
	(* status data structure *)
	Status			: 	ST_AxisStatus;	(* V *)
END_VAR
VAR
END_VAR
IF Enable THEN
	Busy := TRUE;

	Axis.ReadStatus();
	Status := Axis.Status;

	Error			:= 	Status.Error;
	ErrorID			:= 	Status.ErrorID;

	(* motion control statemachine states: *)
	ErrorStop		:= 	Status.ErrorStop;
	Disabled			:= 	Status.Disabled;
	Stopping			:= 	Status.Stopping;
	StandStill		:= 	Status.StandStill;
	DiscreteMotion	:= 	Status.DiscreteMotion;
	ContinuousMotion	:= 	Status.ContinuousMotion;
	SynchronizedMotion:= 	Status.SynchronizedMotion;
	Homing			:= 	Status.Homing;

	(* additional status *)
	ConstantVelocity	:= 	Status.ConstantVelocity;
	Accelerating		:= 	Status.Accelerating;
	Decelerating		:= 	Status.Decelerating;

	Valid := TRUE;
ELSE
	Busy := FALSE;
	Valid := FALSE;
	Error := FALSE;	(* reset at falling edge of Execute *)
	ErrorID := 0;
END_IF
END_FUNCTION_BLOCK

(* POU MC_ReadStopInfo, ST *)
FUNCTION_BLOCK MC_ReadStopInfo
(*	This Function Block returns time and distance that is required
	to stop an axis from its current dynamical state using the 
	parameterized deceleration and jerk values.
	(No motion is actually commanded by this funciton block)
*)
VAR_IN_OUT
	Axis				:	AXIS_REF;	(* B *)
END_VAR
VAR_INPUT
	Execute			:	BOOL;	(* B *)
	Deceleration		:	LREAL;	(* E *)
	Jerk				:	LREAL;	(* E *)
END_VAR
VAR_OUTPUT
	Done 		: 	BOOL;	(* B *)
	Busy		: 	BOOL;	(* E *)
	Error 		: 	BOOL;	(* B *)
	ErrorID 		: 	UDINT;	(* E *)
	StopDistance : 	LREAL;	(* distance required to stop the axis *)
	StopTime	: 	LREAL;	(* time required to stop the axis *)
END_VAR
VAR
	TriggerExecute: R_TRIG;
	state: _E_TcMC_STATES := STATE_INITIALIZATION;
	stStopInfoRequest 	: 	_ST_TcNC_StopInfoRequest;
	stStopInfoResponse 	: 	_ST_TcNC_StopInfoResponse;
	fbAdsReadWrite		: 	ADSRDWRT;
END_VAR
TriggerExecute(CLK:=Execute);

CASE state OF
	STATE_INITIALIZATION:
		IF NOT Execute THEN
			Done := FALSE;
			Error := FALSE;	(* reset at falling edge of Execute *)
			ErrorID := 0;
		END_IF
		IF TriggerExecute.Q THEN
			Done := FALSE;
			Busy := TRUE;
			Error := FALSE;
			ErrorID := 0;
			StopDistance := 0 ;
			StopTime := 0 ;
			stStopInfoRequest.Deceleration := Deceleration;
			stStopInfoRequest.Jerk := Jerk;
			fbAdsReadWrite(WRTRD:=FALSE);
		END_IF
		IF Busy THEN
			fbAdsReadWrite(
				NETID:= TcMcGlobal.NCNETID_TCMC,
				PORT:= TcMcGlobal.NCPORT_TCMC,
				IDXGRP:=TcMcGlobal.Axis.State.IDXGRP+Axis.NcToPlc.AxisId,
				IDXOFFS:= TcMcGlobal.Axis.State.IDXOFFS.STOPINFORMATION,
				WRITELEN:= SIZEOF(stStopInfoRequest),
				READLEN:= SIZEOF(stStopInfoResponse),
				SRCADDR:= ADR(stStopInfoRequest),
				DESTADDR:= ADR(stStopInfoResponse),
				WRTRD:= TRUE,
				TMOUT:= TcMcGlobal.tADSTimeOut );
			IF NOT fbAdsReadWrite.BUSY THEN
				Error := fbAdsReadWrite.ERR;
				ErrorID := fbAdsReadWrite.ERRID;
				Done := NOT Error;
				IF Done THEN
					StopDistance := stStopInfoResponse.StopDistance;
					StopTime := stStopInfoResponse.StopTime;
				END_IF
				Busy := FALSE;
			END_IF
		END_IF
END_CASE
END_FUNCTION_BLOCK

(* POU MC_Reset, ST *)
FUNCTION_BLOCK MC_Reset
(*
	This Function Block makes the transition from the state ErrorStop to StandStill
	or ‘Disabled’ by resetting all internal axis-related errors. It does not affect the 
	output of the FB instances.
*)
VAR_IN_OUT
	Axis				:	AXIS_REF;	(* B *)
END_VAR
VAR_INPUT
	Execute			:	BOOL;		(* B *)
END_VAR
VAR_OUTPUT
	Done			:	BOOL;		(* B *)
	Busy			:	BOOL;		(* E *)
	Error			:	BOOL;		(* B *)
	ErrorID			:	UDINT;		(* B *)
END_VAR
VAR
	ADSbusy		: 	BOOL;
	iState			:	_E_TcMC_STATES := STATE_INITIALIZATION;
	LastExecutionResult: 	_ST_FunctionBlockResults;
END_VAR
{library private}
VAR
	fbAdsWrite		:	_TcMC_ADSWRITE;	(* 2010-05-31 KSt *)
(*	fbAdsWrite		:	ADSWRITE; *)		(* 2010-05-31 KSt *)
	fbOnTrigger		:	R_TRIG;
END_VAR
fbOnTrigger(CLK:= Execute);

CASE iState OF
	STATE_INITIALIZATION: (* initial iState *)
		Busy := FALSE;
		IF NOT Execute THEN
			Done := FALSE;
			Error := FALSE;			(* reset at falling edge of Execute *)
			ErrorID := 0;
		END_IF
		IF fbOnTrigger.Q THEN
			Busy := TRUE;
			Done:= FALSE;
			Error := FALSE;
			ErrorID := 0;
(*			fbAdsWrite(WRITE:=FALSE);*)			(* 2010-05-31 KSt *)
			fbAdsWrite(WRITE:=FALSE, Axis:=Axis);	(* 2010-05-31 KSt *)

			fbAdsWrite(	NETID:= TcMcGlobal.NCNETID_TCMC,
						PORT:= TcMcGlobal.NCPORT_TCMC,
						IDXGRP:=TcMcGlobal.Axis.Functions.IDXGRP+Axis.NcToPlc.AxisId,
						IDXOFFS:= TcMcGlobal.Axis.Functions.IDXOFFS.RESET,
						LEN:= 0,
						SRCADDR:= 0 ,
						WRITE:=TRUE ,
						TMOUT:= TcMcGlobal.tADSTimeOut,
						Axis:=Axis		(* 2010-05-31 KSt *)
					);
			iState := STATE_ORDER;
		END_IF;

	STATE_ORDER:
(*		fbAdsWrite();*)			(* 2010-05-31 KSt *)
		fbAdsWrite( Axis:=Axis );	(* 2010-05-31 KSt *)
		 IF NOT fbAdsWrite.Busy THEN
			IF fbAdsWrite.Err THEN
				ErrorID := fbAdsWrite.ErrId;
				Error := TRUE;
			ELSE
				ErrorID := Axis.NcToPlc.ErrorCode;
				Error := ErrorID <> 0;
				Done := NOT Error;
			END_IF;
(*			fbAdsWrite(WRITE:=FALSE);*)			(* 2010-05-31 KSt *)
			fbAdsWrite(WRITE:=FALSE, Axis:=Axis );	(* 2010-05-31 KSt *)
			Axis.PlcToNc.PlcCycleControl.1 := 0; (* KSt - 2009-08 - reset exceeded flag for external set point generator *)
			iState := STATE_INITIALIZATION;
		END_IF

	ELSE  (* CASE : Unknown program state *)
		Error := TRUE;
		ErrorID := 16#FFFFFFFF;
		iState:= STATE_INITIALIZATION;
END_CASE;

ADSbusy := fbAdsWrite.BUSY;

IF iState=STATE_INITIALIZATION THEN
	(* reset Busy immediately  when sequence ends *)
	IF Busy THEN
		LastExecutionResult.Done := Done;
		LastExecutionResult.Error := Error;
		LastExecutionResult.ErrorID := ErrorID;
	END_IF
	Busy := FALSE;
END_IF
END_FUNCTION_BLOCK

(* POU MC_SetAcceptBlockedDriveSignal, ST *)
FUNCTION MC_SetAcceptBlockedDriveSignal : BOOL
(* 	reference: 	PLC -> NC axis interface (128 bytes)
	copy the signal to bit 8 of an axis nDeCtrlDWord:

	- Accept blocked drive (accept that drive does not follow the controllers
	set point values - e. g. when homing on the limit switches)

	- Akzeptiere blockierten Antrieb (akzeptiere, dass der Antrieb den  
 	Sollwertennicht folgt - z. B. beim Referenzieren auf Endschalter)
*)
VAR_IN_OUT
	Axis				: AXIS_REF;
END_VAR
VAR_INPUT
	Enable : BOOL;
END_VAR
VAR
END_VAR
Axis.PlcToNc.ControlDWord.8 := Enable;
MC_SetAcceptBlockedDriveSignal := Enable;
END_FUNCTION

(* POU MC_SetEncoderScalingFactor, ST *)
FUNCTION_BLOCK MC_SetEncoderScalingFactor
(*
	This function can change the encoder scaling factor in stand-still or on the fly.
*)
VAR_IN_OUT
	Axis			:	AXIS_REF;	(* B *)	(* Identifies the axis to work upon *)
END_VAR
VAR_INPUT
	Execute		:	BOOL;		(* B *)	(* Start setting position in axis *)
	ScalingFactor	:	LREAL;		(* B *)	(* Position unit [u] / EncoderIncrements *)
	Mode		: 	E_SetScalingFactorMode;	(* E *)
	Options		:	ST_SetEncoderScalingOptions;	(* V *)	(* Beckhoff proprietary input *)
END_VAR
VAR_OUTPUT
	Done		:	BOOL;		(* B *)	(* Position has new value *)
	Busy		:	BOOL;		(* E *)	(* Shows that the Function Block is not finished *)
	Error		:	BOOL;		(* B *)	(* Signals that an error has occurred within the Function Block *)
	ErrorID		:	UDINT;		(* E *)	(* Error identification *)
END_VAR
(*
	Note:
	RELATIVE means that the actual position of the axis is adjusted to the 
	new scaling factor value in a way that no position jump will occur.
	ABSOLUTE means that the scaling factor will be set without any 
	internal position offsets. In this case the actual position value of the 
	axis will jump instantaneously.
	When changing the scaling factor on the fly, RELATIVE mode is 
	supposed to be preferred.
*)
VAR
	ADSbusy	: 	BOOL;
	stSetEncoderSaclingFactor	:	_ST_TcNC_SetEncoderSaclingFactor;
	iState		:	_E_TcMC_STATES := STATE_INITIALIZATION;
	fbAdsWrite	:	ADSWRITE;
END_VAR
{library private}
VAR
	fbOnTrigger	:	R_TRIG;
END_VAR
fbOnTrigger(CLK:= Execute);

CASE iState OF
STATE_INITIALIZATION:
	Busy := FALSE;
	IF NOT Execute THEN
		Done := FALSE;
		Error := FALSE;			(* reset at falling edge of Execute *)
		ErrorID := 0;
	END_IF
	IF fbOnTrigger.Q THEN
		Busy := TRUE;
		(* initialize output values *)
		Done := FALSE;
		Error := FALSE;
		ErrorID := 0;
		fbAdsWrite(WRITE := FALSE);

		(* fill structure*)
		stSetEncoderSaclingFactor.fEncoderScalingFactor := ScalingFactor;
		stSetEncoderSaclingFactor.nEncoderScalingFactorType := Mode;
		stSetEncoderSaclingFactor.nCtrlWord.1 := SEL( Options.SelectEncoderIndex, FALSE, TRUE ); 	(* set bit 1 to explicitly select an encoder / control loop - KSt 2009-04-09 *)

		IF Options.SelectEncoderIndex THEN (* KSt 2009-04-09 *)
			(* select the user defined encoder/control loop explicitly *)
			fbAdsWrite.IDXOFFS:= TcMcGlobal.Axis.Functions.IDXOFFS.SETENCODERSCALING + Options.EncoderIndex * 16#00100000;
		ELSE
			(* select the encoder / control loop that is defined by the AXIS_REF interface
				0  	=  select active encoder / control loop		- used when standard AXIS_REF interface is used
				1..n 	=  explicit encoder / control loop selection 	- used when dedicated encoder AXIS_REF interface is used 		*)
			fbAdsWrite.IDXOFFS:= TcMcGlobal.Axis.Functions.IDXOFFS.SETENCODERSCALING + Axis.NcToPlc.ControlLoopIndex * 16#00100000;
		END_IF

		fbAdsWrite(	NETID:= TcMcGlobal.NCNETID_TCMC,
					PORT:= AMSPORT_R0_NCSAF,
					IDXGRP:=TcMcGlobal.Axis.Functions.IDXGRP+Axis.NcToPlc.AxisId,
(*					IDXOFFS:= TcMcGlobal.Axis.Functions.IDXOFFS.SETENCODERSCALING + Options.EncoderIndex * 16#100000,*) (* KSt 2009-04-09 - see selection above *)
					LEN:= SIZEOF(stSetEncoderSaclingFactor),
					SRCADDR:= ADR(stSetEncoderSaclingFactor),
					WRITE:= TRUE,
					TMOUT:= TcMcGlobal.tADSTimeOut);
		iState := STATE_ORDER;
	END_IF;

STATE_ORDER:
	fbAdsWrite();
	IF NOT fbAdsWrite.Busy THEN
		IF fbAdsWrite.Err THEN
			ErrorID := fbAdsWrite.ErrId;
			Error := TRUE;
		ELSE
			Done := TRUE;
		END_IF;
		fbAdsWrite(WRITE := FALSE);
		iState := STATE_INITIALIZATION;
	END_IF;

ELSE  (* CASE : Unknown program state *)
	Error := TRUE;
	ErrorID := 16#FFFFFFFF;
	iState:= STATE_INITIALIZATION;
END_CASE

ADSbusy := fbAdsWrite.BUSY;

IF iState=STATE_INITIALIZATION THEN
	(* reset Busy immediately  when sequence ends *)
	Busy := FALSE;
END_IF
END_FUNCTION_BLOCK

(* POU MC_SetOverride, ST *)
FUNCTION_BLOCK MC_SetOverride
(*
	This Function Block sets the values of override for the whole axis, and all functions 
	that are working on that axis. The override parameters contribute as a factor to the 
	calculation of the commanded velocity, acceleration and jerk of the motion.
*)
VAR_IN_OUT
	Axis			:	AXIS_REF;
END_VAR
VAR_INPUT
	Enable		:	BOOL;	(* B *)
	VelFactor	:	LREAL	(* B *)	:= 1.0;	(* 1.0 = 100% *)
	AccFactor	:	LREAL	(* E *)	:= 1.0;	(* 1.0 = 100% *)	(* not supported *)
	JerkFactor	:	LREAL 	(* E *)	:= 1.0;	(* 1.0 = 100% *)	(* not supported *)
END_VAR
VAR_OUTPUT
	Enabled		:	BOOL;	(* B *)
	Busy		:	BOOL;	(* E *)
	Error		:	BOOL;	(* B *)
	ErrorID		:	UDINT;	(* E *)
END_VAR
(*
	Notes:
	1. The Input AccFactor acts on positive and negative acceleration (deceleration).
	2. This Function Block sets the factor. The override factor is valid until a new override is set.
	3. The default values of the override factor are 1.0.
	4. The value of the overrides can be between 0.0 and 1.0. The behavior of values > 1.0 is 
	     vendor specific. Values< 0.0 are not allowed. The value 0.0 is not allowed for ‘AccFactor’ 
	     and ‘JerkFactor’.
	5. The value 0.0 set to the ‘VelFactor’ stops the axis without bringing it to the state ‘Standstill’.
	6. Override does not act on slave axes. (Axes in the state synchronized motion).
	7. The Function Block does not influence the state diagram of the axis.
	8. ‘VelFactor’ can be changed at any time and acts directly on the ongoing motion.
	9. If in ‘Discrete’ motion, reducing the ‘AccFactor’ and/or ‘JerkFactor’ can lead to a position 
	     overshoot – a possible cause of damage
	10. Activating this Function Block on an axis that is under control of MC_PositionProfile, 
	     MC_VelocityProfile, or MC_AccelerationProfile, is vendor specific.
*)
VAR
END_VAR
IF Enable THEN
	Busy := TRUE;
	IF VelFactor > 1 OR VelFactor < 0 THEN
		ErrorID := MC_ERROR_PARAMETER_NOT_CORRECT;
		Error := TRUE;
	ELSE
		Axis.PlcToNc.Override := LREAL_TO_UDINT(VelFactor*1000000);
		ErrorID := MC_ERROR_NO_ERROR;
		Error := FALSE;
		Enabled:=TRUE;
	END_IF;
ELSE
	Busy := FALSE;
	Enabled:=FALSE;
	Error := FALSE;			(* reset at falling edge of Execute *)
	ErrorID := 0;
END_IF;
END_FUNCTION_BLOCK

(* POU MC_TableBasedPositionCompensation, ST *)
(*==============================================================================*)
(* Name:	MC_TableBasedPositionCompensation										*)
(*		(based on _FB_PositionCorrectionTableLookup + MC_PositionCorrectionLimiter)	*)
(* Parameter: returns a compensation value depending on the position of the reference axis	*)
(*		Use the nc function PositionCompensation to compensate a position error			*)
(*		1. the FB _FB_PositionCorrectionTableLookup calculates the correction value		*)
(*		2. the FB MC_PositionCorrectionLimiter feed this correction value					*)
(*		into the NcToPlc.PositionCorrection variable									*)
(* Author:	 	HKP																	*)
(* Date:		19-July-2012															*)
(* last edit:	VER 0.0.4															*)
(*==============================================================================*)
FUNCTION_BLOCK MC_TableBasedPositionCompensation
VAR_IN_OUT
	Axis							: Axis_Ref;
END_VAR
VAR_INPUT
	Enable						: BOOL; 				(* rising edge triggers initialize routine *)
	pTable						: POINTER TO ST_PositionCompensationTableElement;	(* pointer to equidistant table with strictly monotonous increasing position values *)
	TableSize					: UDINT;				(* size of data in bytes related to 'pTable' *)
	TableParameter				: ST_PositionCompensationTableParameter;	(* position compensation table parameter structure *)
	Ramp						: LREAL;								(* velocity limit for feeded position compensation (constant velocity and linear position sub profile for position compensation) [mm/s] (default:=0.0) *)
	DisableMode					: E_DisableMode;						(* disable mode defines whow to react in case of disabling: (0)=HOLD, (1)=RESET, ... *)
	Options						: ST_PositionCompensationOptions;		(* optional parameters (NOT USED YET) *)
END_VAR
VAR_OUTPUT
	Enabled						: BOOL;
	Busy						: BOOL;
	Error						: BOOL;
	ErrorID						: UDINT;
	CurrentCorrection				: LREAL;								(* current actual position correction value [mm] *)
	Limiting						: BOOL;								(* function block is currently limiting the Position Correction *)
END_VAR
VAR
	InternalEnable				: BOOL;								(* trick for internal FB handling *)
	state						: INT;
	GetThisTaskIndex				: GETCURTASKINDEX;
	CycleTime					: LREAL;								(* task cycle time [s] *)
	fbCalcPositionCorrection		: _FB_PositionCorrectionTableLookup;	(* based on old 'FB_PositionCompensation' in TcNc.lib *)
	fbFeedPositionCorrection		: MC_PositionCorrectionLimiter;			(* s.TcMC2.lib (original based on old 'FB_WritePositionCorrection' in TcNc.lib) *)
	CalcPosCorrOut				: ST_McOutputs;
	FeedPosCorrOut				: ST_McOutputs;
	InternalAcceleration			: LREAL;								(* input of FB 'MC_PositionCorrectionLimiter': 'Acceleration' [mm/s^2] *)
	InternalCorrectionValue			: LREAL;								(* output of FB 'MC_PositionCorrectionLimiter': 'PositionCorrectionValue' [mm] *)
	InternalLimitingActive			: BOOL;								(* output of FB 'MC_PositionCorrectionLimiter': 'Limiting' [0/1] *)
END_VAR
CASE state OF
	0 : (* init *)
		Busy := FALSE;
		Enabled := FALSE;
		IF Enable THEN
			IF NOT Axis.NcToPlc.OpModeDWord.20 THEN (* PositionCorrection active ? *)
				Error := TRUE;
				ErrorID := MC_ERROR_WRONG_MODE;
				state := 9999;
			ELSIF Ramp < 0 THEN
				Error := TRUE;
				ErrorID := MC_ERROR_PARAMETER_NOT_CORRECT;
				state := 9999;
			ELSE
				Busy := TRUE;
				state := 1;
			END_IF
		END_IF

	1 : (* active *)
		Enabled := TRUE;


		(* cycle time needed for pre calculation of the acceleration input *)
		IF CycleTime = 0 THEN
			GetThisTaskIndex;
			CycleTime := SystemTaskInfoArr[GetThisTaskIndex.index].cycleTime * LREAL#100E-9;
		END_IF

		(* special handling for disabling (depends from disable mode) *)
		IF( Enable = FALSE ) THEN
			(* disable mode HOLD *)
			IF( (DisableMode = DisableModeHold) ) THEN
				InternalEnable := TRUE;
				IF( Ramp > 0.0 ) THEN
					InternalAcceleration := Ramp / CycleTime;			(* mm/s^2 = mm/s / s *)
				ELSE
					InternalAcceleration := 0.0;
				END_IF
			(* disable mode RESET *)
			ELSE
				InternalEnable := Enable;
				InternalAcceleration := 0.0;
			END_IF
		(* active *)
		ELSE
			InternalEnable := Enable;
			IF( Ramp > 0.0 ) THEN
				InternalAcceleration := Ramp / CycleTime;			(* mm/s^2 = mm/s / s *)
			ELSE
				InternalAcceleration := 0.0;
			END_IF
		END_IF


		(* 1.) calculate position correction (if enabled) *)
		(* '_FB_PositionCorrectionTableLookup' *)
		fbCalcPositionCorrection(
		   (* Enable := Enable, *)
		   Enable := InternalEnable,
		   pTable := pTable,
		   TableSize := TableSize,
		   Axis := Axis,
		   TableParameter := TableParameter,
		   Compensation => InternalCorrectionValue,
		   Error => CalcPosCorrOut.Error,
		   ErrorId => CalcPosCorrOut.ErrorID,
		   Active => CalcPosCorrOut.Active );

		(* check for error return code *)
		IF CalcPosCorrOut.Error THEN
			Error := TRUE;
			ErrorID := CalcPosCorrOut.ErrorID;
			state := 9999;
		END_IF


		(* 2.) feed position compensation (acceleration limited, that means linear velocity ramp) *)
		(*
				POSITIONCORRECTIONMODE_FAST
					The limitatation to maximum position change per cycle. Due to the maximum 
					change per cycle, the correction will take place as fast as possible and may 
					also be unlimited if PositionCorrectionValue is changed slightly. 
		*)
		(* MC_PositionCorrectionLimiter *)
		fbFeedPositionCorrection(
		(*	Enable :=TRUE, *)
			 Enable :=Enable,
			 PositionCorrectionValue := InternalCorrectionValue,
			 CorrectionMode := POSITIONCORRECTION_MODE_FAST,
			 Acceleration := InternalAcceleration,			(* HKP: pre calculated internal acceleration limit *)
			 CorrectionLength := 0.0,					(* optional length - not used for this correction mode 'POSITIONCORRECTION_MODE_FAST' *)
			 Axis := Axis,
			 Busy => FeedPosCorrOut.Busy,
			 Error => FeedPosCorrOut.Error,
			 ErrorID =>FeedPosCorrOut.ErrorID,
			 Limiting => InternalLimitingActive
			);

		(* check for error return code *)
		IF FeedPosCorrOut.Error THEN
			Error := TRUE;
			ErrorID := FeedPosCorrOut.ErrorID;
			state := 9999;
		END_IF


		CurrentCorrection	:= InternalCorrectionValue;
		Limiting			:= InternalLimitingActive;

		IF NOT Enable THEN
			Enabled := FALSE;
			state := 0;
		END_IF

	9999 : (* error *)
		IF NOT Enable THEN
			Error := FALSE;
			ErrorID := 0;
			state := 0;
		END_IF
END_CASE

IF state = 0 THEN
	Busy := FALSE;
END_IF
END_FUNCTION_BLOCK

(* POU MC_TouchProbe, ST *)
FUNCTION_BLOCK MC_TouchProbe
(*
	The function block is used to record an axis position at a trigger event

	Notes:
	1. Intended for single shot operation, that is the first event after the rising edge at ‘Execute’ 
	     is valid for recordingonly. Possible following events are ignored
	2. One Function Block instance should represent exactly one probing command

*)
VAR_IN_OUT
	Axis				:	AXIS_REF; 		(* B *)	(* Identifies the axis which position should be recorded at a defined event at the trigger input *)
	TriggerInput		: 	TRIGGER_REF; 	(* B *)	(* Reference to the trigger signal source. *)
END_VAR
VAR_INPUT
	Execute			:	BOOL;	(* B *)	(* Starts touch probe recording *)
	WindowOnly		: 	BOOL;	(* E *)	(* Enables the monitoring window *)
	FirstPosition		: 	LREAL;	(* E *)	(* Beginning of the monitoring window *)
	LastPosition		: 	LREAL;	(* E *)	(* Ending of the monitoring window *)
END_VAR
VAR_OUTPUT
	Done			:	BOOL;	(* B *)	(* move completed *)
	Busy			: 	BOOL;	(* E *)	(* function block is currently Busy *)
	CommandAborted	: 	BOOL;	(* E *)
	Error			:	BOOL;	(* B *)	(* Signals that error has occurred within Function Block *)
	ErrorID			:	UDINT;	(* E *)	(* Error identification *)
	RecordedPosition:	LREAL;	(* B *)	(* Position where trigger event occurred *)
END_VAR
VAR
	ADSbusy: BOOL;
	iState			: 	_E_TcMC_STATES := STATE_INITIALIZATION;
	TouchProbeValid	: 	ARRAY[1..4] OF UDINT;	(* valid state of probes 1..4 *)
	TouchProbeActive: 	ARRAY[1..4] OF UDINT;	(* activation state of probes 1..4 *)
	TouchProbeValue : 	ARRAY[1..4] OF LREAL;	(* last recorded value of probes 1..4 *)
	TouchProbeModuloValue : 	ARRAY[1..4] OF LREAL;	(* last recorded modulo value of probes 1..4 *)
	TouchProbeInactiveCounter: 	ARRAY[1..4] OF INT;	(* number of cycles where the probes 1..4 where inactive (activation monitoring) *)
END_VAR
{library private}
VAR CONSTANT
	OLDADSINTERFACE : BOOL := TRUE; (* temporary flag to test old and new NC ADS touch probe interface *)
END_VAR
VAR
	fbADSwrite		: 	ADSWRITE;
	fbAdsReadValid	: 	ADSREAD;
	fbAdsReadValue	: 	ADSREAD;
	fbAdsReadState	: 	ADSREAD;
	fbAdsReadModulo: 	ADSREAD;
	TimerAdsReadState: 	TON;
	RtrigPlcEvent		: 	R_TRIG;
	FtrigPlcEvent		: 	F_TRIG;
	fbOnTrigger		: 	R_TRIG;
	LatchID			: 	UDINT;
	Restart			: 	BOOL;	(* restart probe sequence when the trigger was outside the defined window *)
	InWindow		: 	BOOL;	(* probe value is inside the defined window *)
	ModuloFactor		: 	LREAL;	(* axis' modulo factor read from the NC *)
	InitDone			: 	BOOL;	(* initialization on start-up finished *)
	IndexOffset		: 	WORD;
	i: INT;
END_VAR
 fbOnTrigger(CLK:= Execute);

CASE iState OF
	STATE_INITIALIZATION :
		Busy := FALSE;
		IF NOT Execute THEN
			Done := FALSE;
			Error := FALSE;			(* reset at falling edge of Execute *)
			ErrorID := 0;
		END_IF

		ActTouchProbeStartupInit();	(* will return InitDone *)

		IF fbOnTrigger.Q THEN
			Restart := TRUE;
		END_IF

		IF Restart THEN
			(* check initialization *)
			Busy := fbAdsReadModulo.BUSY;
			Error := fbAdsReadModulo.ERR;
			ErrorID := fbAdsReadModulo.ERRID;
			IF NOT Busy AND NOT InitDone THEN
				(* initialization error *)
				fbAdsReadModulo(READ:=FALSE);	(* initialize again during next cycle *)
				Restart := FALSE;	(* error *)
			ELSIF InitDone THEN;
				Busy := TRUE;
				IF NOT fbADSwrite.BUSY THEN
					(* initialization *)
					Done := FALSE;
					Error := FALSE;
					ErrorID := 0;
					CommandAborted := FALSE;
					RecordedPosition := 0;
					fbADSwrite(WRITE:=FALSE); (* reset *)
					fbAdsReadValid(READ:=FALSE);
					fbAdsReadValue(READ:=FALSE);
					fbAdsReadState(READ:=FALSE);
					TimerAdsReadState(IN:=FALSE);
					RtrigPlcEvent(CLK:=TriggerInput.PlcEvent);
					FtrigPlcEvent(CLK:=TriggerInput.PlcEvent);
					Restart := FALSE;
					FOR i := 1 TO 4 DO
						TouchProbeInactiveCounter[i] := 0;
					END_FOR
				END_IF

				CASE TriggerInput.Edge OF
					RisingEdge :
						IndexOffset := 16#201;
					FallingEdge:
						IndexOffset := 16#202;
				ELSE (* case *)
					Error := TRUE;
					ErrorID := MC_ERROR_INVALID_TOUCH_PROBE;
				END_CASE

				IF TriggerInput.EncoderID > 255 THEN
					Error := TRUE;
					ErrorID := MC_ERROR_INVALID_TOUCH_PROBE;
				END_IF

				IF NOT Error THEN
					CASE TriggerInput.TouchProbe OF
						TouchProbe1,
						TouchProbe2,
						TouchProbe3,
						TouchProbe4:
							(* activate latch *)
							ActTouchProbeActivate();
							iState := STATE_ORDER;

						PlcEvent:
							(* no action necessary here *);
							TriggerInput.ProbeState := TouchProbeActivated;
							iState := STATE_WAITING;
					ELSE
						Error := TRUE;
						ErrorID := MC_ERROR_INVALID_TOUCH_PROBE;
					END_CASE
				END_IF
			END_IF
		END_IF

	STATE_ORDER :	(* wait until probe is activated *)
		ActTouchProbeActivate();

	STATE_WAITING : (* wait until touch probe was trigerred *)
		CASE TriggerInput.TouchProbe OF (* type of touch probe *)
			TouchProbe1,
			TouchProbe2,
			TouchProbe3,
			TouchProbe4:
				ActTouchProbeMonitorLatchValid();
				IF iState=STATE_WAITING THEN (* still not triggered *)
					ActTouchProbeMonitorActivity();
				END_IF

			(* CASE PlcEvent *)
			PlcEvent : (* touch proble will be triggered through a PLC signal (TriggerInput.PlcEvent) *)
				ActTouchProbeMonitorPlcEvent();
		END_CASE (* type of touch probe *)

		IF NOT Done AND (TriggerInput.ProbeState = TouchProbeAborted) THEN
			(* function block has been aborted by an external MC_AbortTrigger *)
			CommandAborted := TRUE;
			iState := STATE_INITIALIZATION;
		END_IF

		IF iState<> STATE_WAITING THEN
			(* leave the waiting state now *)
			TriggerInput.ProbeState := TouchProbeInactive;
			fbAdsReadModulo(READ:=FALSE);	(* initialize again during next cycle *)
		END_IF
END_CASE

ADSbusy := fbAdsWrite.BUSY OR fbAdsReadValid.BUSY OR fbAdsReadValue.BUSY OR fbAdsReadState.BUSY OR fbAdsReadModulo.BUSY;
IF iState=STATE_INITIALIZATION AND NOT Restart THEN
	(* reset Busy immediately  when sequence ends *)
	Busy := FALSE;
END_IF
END_FUNCTION_BLOCK
ACTION ActTouchProbeActivate:
(* start the touch probe sequence *)

LatchID := TriggerInput.TouchProbe;
TriggerInput.ProbeState := TouchProbeActivated;

fbADSwrite(	NETID:= TcMcGlobal.NCNETID_TCMC,
			PORT:=AMSPORT_R0_NCSAF ,
			IDXGRP:=16#5200+TriggerInput.EncoderID ,
			IDXOFFS:=IndexOffset,
			LEN:=SEL(OLDADSINTERFACE, SIZEOF(LatchID), 0) ,
			SRCADDR:=ADR(LatchID),
			WRITE:=TRUE ,
			TMOUT:=TcMcGlobal.tADSTimeOut);

IF NOT fbADSwrite.BUSY THEN
	IF fbADSwrite.ERR THEN
		Error := fbADSwrite.ERR;
		ErrorID := fbADSwrite.ERRID;
	END_IF
	IF NOT Error AND TriggerInput.ProbeState = TouchProbeAborted THEN
		(* Synchronization error between MC_TouchProbe and MC_AbortTrigger *)
		Error := TRUE;
		ErrorID := MC_ERROR_TOUCH_PROBE_DEACTIVATED;
	END_IF
	TriggerInput.ProbeState := SEL( Error, TouchProbeActivated, TouchProbeInactive );
	iState := SEL( Error, STATE_WAITING, STATE_INITIALIZATION);
END_IF
END_ACTION
ACTION ActTouchProbeMonitorActivity:
(* check if latch is still active *)
TimerAdsReadState(IN := NOT TimerAdsReadState.q , PT:=T#1s);
IF TimerAdsReadState.q OR fbAdsReadState.BUSY THEN
	fbAdsReadState(	NETID:= TcMcGlobal.NCNETID_TCMC,
				PORT:=AMSPORT_R0_NCSAF ,
				IDXGRP:=16#5100+TriggerInput.EncoderID ,
				IDXOFFS:= 16#201,
				LEN:=SEL(OLDADSINTERFACE, SIZEOF(TouchProbeActive), 2),
				DESTADDR:=ADR(TouchProbeActive) ,
				READ:=TRUE ,
				TMOUT:=TcMcGlobal.tADSTimeOut );
	IF NOT fbAdsReadState.BUSY THEN
		IF fbAdsReadState.ERR THEN
			Error := TRUE;
			ErrorID := fbAdsReadState.ERRID;
		ELSE
			IF TouchProbeActive[TriggerInput.TouchProbe]<>1 THEN
				TouchProbeInactiveCounter[TriggerInput.TouchProbe] := TouchProbeInactiveCounter[TriggerInput.TouchProbe] + 1;
				IF TouchProbeInactiveCounter[TriggerInput.TouchProbe] > 1 THEN
					(* error condition when the probing sequence is inactive more than once *)
					Error := TRUE;
					ErrorID := MC_ERROR_TOUCH_PROBE_DEACTIVATED;
					CommandAborted := TRUE;
					iState := STATE_INITIALIZATION;
				END_IF
			END_IF
		END_IF
		fbAdsReadState(READ:=FALSE); (* reset *)
	END_IF
END_IF
END_ACTION
ACTION ActTouchProbeMonitorLatchValid:
(* monitor if the touch probe has been triggered *)

IF F_AxisExternalLatchValid(Axis.NcToPlc.StateDWord) THEN
	(* read the status of the latch *)
	fbAdsReadValid(	NETID:= TcMcGlobal.NCNETID_TCMC,
				PORT:=AMSPORT_R0_NCSAF ,
				IDXGRP:=16#5100+TriggerInput.EncoderID ,
				IDXOFFS:= 16#202,
				LEN:=SEL(OLDADSINTERFACE, SIZEOF(TouchProbeValid), 2) ,
				DESTADDR:=ADR(TouchProbeValid) ,
				READ:=TRUE ,
				TMOUT:=TcMcGlobal.tADSTimeOut );
	(* read the latched value *)
	fbAdsReadValue(	NETID:= TcMcGlobal.NCNETID_TCMC,
				PORT:=AMSPORT_R0_NCSAF ,
				IDXGRP:=16#5100+TriggerInput.EncoderID ,
				IDXOFFS:= 16#205,
				LEN:=SEL(OLDADSINTERFACE, SIZEOF(TouchProbeValue), SIZEOF(TouchProbeValue[1])) ,
				DESTADDR:=ADR(TouchProbeValue) ,
				READ:=TRUE ,
				TMOUT:=TcMcGlobal.tADSTimeOut );
	IF NOT fbAdsReadValid.BUSY AND NOT fbAdsReadValue.BUSY THEN
		IF fbAdsReadValid.err THEN
			Error := TRUE;
			ErrorID := fbAdsReadValid.ERRID;
			iState := STATE_INITIALIZATION;
		ELSIF fbAdsReadValue.err THEN
			Error := TRUE;
			ErrorID := fbAdsReadValue.ERRID;
			iState := STATE_INITIALIZATION;
		ELSE (* no error *)
			IF TouchProbeValid[TriggerInput.TouchProbe]=1 THEN
				RecordedPosition:=TouchProbeValue[TriggerInput.TouchProbe];
				Done := TRUE;
				IF TriggerInput.ModuloPositions AND (ModuloFactor<>0) THEN	(* check for  (ModuloFactor=0) - 2007-02-06 KSt *)
(*					RecordedPosition :=  ((RecordedPosition / ModuloFactor) - TRUNC(RecordedPosition / ModuloFactor)) * ModuloFactor;*)	(* 20101027 KSt *)
					RecordedPosition := MODABS(RecordedPosition,  ModuloFactor);	(* 20101027 KSt *)
					TouchProbeModuloValue[TriggerInput.TouchProbe] := RecordedPosition;
(*					InWindow := (RecordedPosition>=FirstPosition) AND (RecordedPosition<=LastPosition);*)	(* 20110216 KSt *)
					IF FirstPosition>LastPosition THEN (* 20110216 KSt *)
						InWindow := (RecordedPosition>=FirstPosition) OR  (RecordedPosition<=LastPosition);  (* 20110216 KSt *)
					ELSE
						InWindow := (RecordedPosition>=FirstPosition) AND (RecordedPosition<=LastPosition);
					END_IF
				ELSE
					InWindow := (RecordedPosition>=FirstPosition) AND (RecordedPosition<=LastPosition);
				END_IF
				IF WindowOnly AND NOT InWindow THEN
					RecordedPosition:=0;
					Done := FALSE;
					Restart := TRUE; (* ignore this event, latch next one *)
				END_IF
				iState := STATE_INITIALIZATION;
			ELSE
				fbAdsReadValid(READ:=FALSE);
				fbAdsReadValue(READ:=FALSE);
			END_IF
		END_IF
	END_IF
END_IF
END_ACTION
ACTION ActTouchProbeMonitorPlcEvent:
(* touch probe sequence for simple PLC inputs *)
(* monitor PLC input trigger *)

RtrigPlcEvent(CLK:=TriggerInput.PlcEvent);
FtrigPlcEvent(CLK:=TriggerInput.PlcEvent);
IF ((TriggerInput.Edge=RisingEdge) AND RtrigPlcEvent.Q) OR
   ((TriggerInput.Edge=FallingEdge) AND FtrigPlcEvent.Q) THEN
	RecordedPosition:=Axis.NcToPlc.ActPos; 	(* 2007-02-06 KSt *)
	IF TriggerInput.ModuloPositions AND (ModuloFactor<>0) THEN	(* check for  (ModuloFactor=0) - 2007-02-06 KSt *)
(*		RecordedPosition :=  ((RecordedPosition / ModuloFactor) - TRUNC(RecordedPosition / ModuloFactor)) * ModuloFactor;*)	(* 20101027 KSt *)
		RecordedPosition :=  MODABS(RecordedPosition,  ModuloFactor);	(* 20101027 KSt *)
(*		InWindow := (RecordedPosition>=FirstPosition) AND (RecordedPosition<=LastPosition);*)	 (* 20110216 KSt *)
		IF FirstPosition>LastPosition THEN (* 20110216 KSt *)
			InWindow := (RecordedPosition>=FirstPosition) OR  (RecordedPosition<=LastPosition);  (* 20110216 KSt *)
		ELSE
			InWindow := (RecordedPosition>=FirstPosition) AND (RecordedPosition<=LastPosition);
		END_IF
	ELSE
		InWindow := (RecordedPosition>=FirstPosition) AND (RecordedPosition<=LastPosition);
	END_IF
	IF WindowOnly AND NOT InWindow THEN
		RecordedPosition:=0;	(* 2007-02-06 KSt *)
	ELSE
		Done := TRUE;
		iState := STATE_INITIALIZATION;
	END_IF
END_IF
END_ACTION
ACTION ActTouchProbeStartupInit:
(* initialization on plc start-up *)
(* read the axis' modulo factor *)

IF TriggerInput.ModuloPositions THEN
	IF ModuloFactor = 0 THEN
		InitDone := FALSE; (* 2007-02-06 KSt *)
	END_IF
	fbAdsReadModulo(	NETID:= TcMcGlobal.NCNETID_TCMC,
						PORT:= AMSPORT_R0_NCSAF,
						IDXGRP:= 16#5000+TriggerInput.EncoderID ,
						IDXOFFS:= 16#9,
						LEN:= SIZEOF(ModuloFactor),
						DESTADDR:= ADR(ModuloFactor),
						READ:= TRUE,
						TMOUT:= TcMcGlobal.tADSTimeOut);
	IF NOT fbAdsReadModulo.BUSY THEN
		IF fbAdsReadModulo.ERR OR (ModuloFactor=0) THEN
			fbAdsReadModulo( READ:=FALSE ); 	(* 2007-02-06 KSt *)
			InitDone := FALSE; 	(* init failed - 2007-02-06 KSt *)
			Error := TRUE;
			ErrorID := fbAdsReadModulo.ERRID;
		ELSE
			InitDone := TRUE;
		END_IF
	END_IF
ELSE (* no modulo positions *)
	fbAdsReadModulo( READ:=FALSE );	(* 2007-02-06 KSt *)
	InitDone := TRUE;
END_IF
END_ACTION

(* POU MC_TouchProbe_V2_00, ST *)
FUNCTION_BLOCK MC_TouchProbe_V2_00
(*	The function block is used to record an axis position at a trigger event *)
VAR_IN_OUT
	Axis				:	AXIS_REF; 		(* B *)	(* Identifies the axis which position should be recorded at a defined event at the trigger input *)
	TriggerInput		: 	TRIGGER_REF; 	(* B *)	(* Reference to the trigger signal source. *)
END_VAR
VAR_INPUT
	Execute			:	BOOL;	(* B *)	(* Starts touch probe recording *)
	WindowOnly		: 	BOOL;	(* E *)	(* Enables the monitoring window *)
	FirstPosition		: 	LREAL;	(* E *)	(* Beginning of the monitoring window *)
	LastPosition		: 	LREAL;	(* E *)	(* Ending of the monitoring window *)
END_VAR
VAR_OUTPUT
	Done			:	BOOL;	(* B *)	(* move completed *)
	Busy			: 	BOOL;	(* E *)	(* function block is currently Busy *)
	CommandAborted	: 	BOOL;	(* E *)
	Error			:	BOOL;	(* B *)	(* Signals that error has occurred within Function Block *)
	ErrorID			:	UDINT;	(* E *)	(* Error identification *)
	RecordedPosition	:	LREAL;	(* B *)	(* Position where trigger event occurred *)
	RecordedData	:	MC_TouchProbeRecordedData;	(* V *)	(* data additional to RecordedPosition *)
END_VAR
VAR
	ADSbusy: BOOL;
	iState			: 	_E_TcMC_STATES := STATE_INITIALIZATION;
	ExternalLatchValid: BOOL;
	TouchProbeValid	: 		ARRAY[1..4] OF UDINT;	(* valid state of probes 1..4 *)
	TouchProbeActive: 		ARRAY[1..4] OF UDINT;	(* activation state of probes 1..4 *)
	TouchProbeValue : 		ARRAY[1..4] OF LREAL;	(* last recorded value of probes 1..4 *)
	TouchProbeModuloValue : 	ARRAY[1..4] OF LREAL;	(* last recorded modulo value of probes 1..4 *)
	TouchProbeCounter : 		ARRAY[1..4] OF UDINT;	(* last recorded value counter of probes 1..4 *)
	TouchProbeInactiveCounter: 	ARRAY[1..4] OF INT;	(* number of cycles where the probes 1..4 where inactive (activation monitoring) *)
	stTouchProbeActivation : _ST_TcNc_TouchProbeActivation;
	stTouchProbeStatusRequest : _ST_TcNc_TouchProbeStatusRequest;
	stTouchProbeStatusResponse : _ST_TcNc_TouchProbeStatusResponse;
	stTouchProbeDeactivation : _ST_TcNc_TouchProbeDeactivation;
END_VAR
{library private}
VAR
	LastTouchProbeValue : 	ARRAY[1..4] OF LREAL;	(* last recorded value of probes 1..4 *)
	LastTouchProbeCounter : 	ARRAY[1..4] OF UDINT;	(* last recorded value counter of probes 1..4 *)
	fbADSwrite		: 	ADSWRITE;
	fbAdsReadValid	: 	ADSREAD;
	fbAdsReadValue	: 	ADSREAD;
	fbAdsReadState	: 	ADSREAD;
	fbAdsReadModulo: 	ADSREAD;
	fbAdsReadLatchStatus: ADSRDWRTEX;
	TimerAdsReadState: 	TON;
	RtrigPlcEvent		: 	R_TRIG;
	FtrigPlcEvent		: 	F_TRIG;
	fbOnTrigger		: 	R_TRIG;
	Restart			: 	BOOL;	(* restart probe sequence when the trigger was outside the defined window *)
	InWindow		: 	BOOL;	(* probe value is inside the defined window *)
	ModuloFactor		: 	LREAL;	(* axis' modulo factor read from the NC *)
	InitDone			: 	BOOL;	(* initialization on start-up finished *)
	IndexOffset		: 	WORD;
	iTriggerInput		: 	TRIGGER_REF; 	(* B *)	(* Reference to the trigger signal source. *)
	i: INT;
END_VAR
(* 	MC_TouchProbe main sequence *)

fbOnTrigger(CLK:= Execute);
ExternalLatchValid := F_AxisExternalLatchValid(Axis.NcToPlc.StateDWord);

CASE iState OF
	STATE_INITIALIZATION :
		Busy := FALSE;
		IF NOT Execute THEN
			Done := FALSE;
			Error := FALSE;			(* reset at falling edge of Execute *)
			ErrorID := 0;
		END_IF

		ActTouchProbeStartupInit();	(* will return InitDone *)

		(* read version of NC *)
		IF TcMcGlobal.NcDeviceInfoNcVersion=0 THEN
			TcMcGlobal.ReadDeviceInfo();
		END_IF
		
		IF fbOnTrigger.Q THEN
			Restart := TRUE;
		END_IF

		IF Restart THEN
			Busy := TRUE;

			(* check initialization *)
			IF NOT InitDone AND NOT fbAdsReadModulo.BUSY AND NOT TcMcGlobal.fbADSRDDEVINFO.BUSY THEN
				(* initialization error *)
				Busy := fbAdsReadModulo.BUSY;
				Error := fbAdsReadModulo.ERR;
				ErrorID := fbAdsReadModulo.ERRID;
				fbAdsReadModulo(READ:=FALSE);	(* initialize again during next cycle *)
				Restart := FALSE;	(* error *)
			ELSIF InitDone AND NOT TcMcGlobal.fbADSRDDEVINFO.BUSY THEN;
				(* initialization was okay - check input parameters *)

				IF NOT fbADSwrite.BUSY THEN
					(* initialization *)
					Done := FALSE;
					Error := FALSE;
					ErrorID := 0;
					CommandAborted := FALSE;
					RecordedPosition := 0;
					fbADSwrite(WRITE:=FALSE); (* reset *)
					fbAdsReadValid(READ:=FALSE);
					fbAdsReadValue(READ:=FALSE);
					fbAdsReadState(READ:=FALSE);
					TimerAdsReadState(IN:=FALSE);
					RtrigPlcEvent(CLK:=TriggerInput.PlcEvent);
					FtrigPlcEvent(CLK:=TriggerInput.PlcEvent);
					LastTouchProbeValue := TouchProbeValue;
					LastTouchProbeCounter := TouchProbeCounter;
					Restart := FALSE;
					FOR i := 1 TO 4 DO
						TouchProbeInactiveCounter[i] := 0;
					END_FOR
				END_IF

